Yaskawa INFORM job: DEMO_ROOF_UPPER_0625_3PAINT_6.JBI

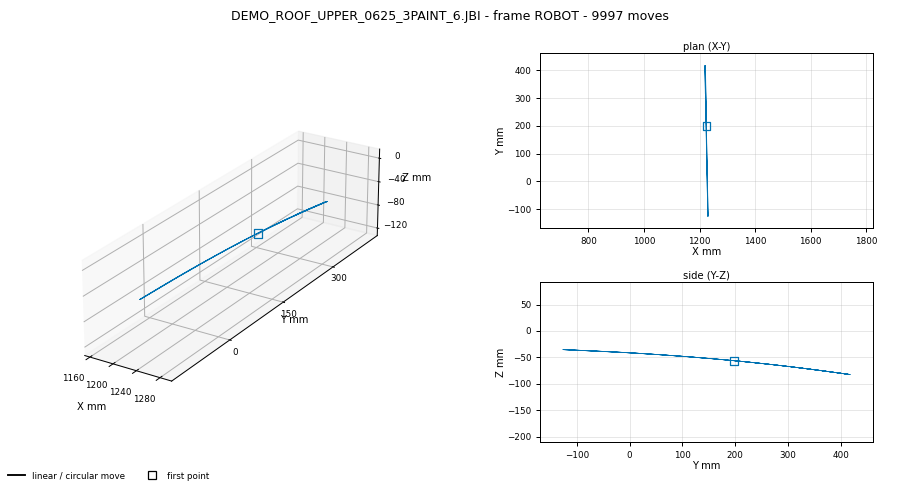
[picture p0: tool path of DEMO_ROOF_UPPER_0625_3PAINT_6.JBI in frame ROBOT, 9997 of 9997 moves have a stored position in this frame; points joined in program order, loops and branches not executed]
/JOB
//NAME DEMO_ROOF_UPPER_0625_3PAINT6
//POS
///NPOS 9997,0,0,0,0,0
///TOOL 0
///USER 0
///POSTYPE ROBOT
///RECTAN
///RCONF 1,0,0,0,0,0,0,0,0,0,0,0,0,0,0,0,0,0,0,0,0,0,0,0
C00000=1225.136,197.844,-56.153,-177.445,6.042,148.322
C00001=1225.132,198.093,-56.176,-177.443,6.043,148.321
C00002=1225.127,198.342,-56.200,-177.440,6.045,148.321
C00003=1225.123,198.590,-56.224,-177.437,6.047,148.321
C00004=1225.118,198.839,-56.247,-177.434,6.049,148.320
C00005=1225.114,199.088,-56.271,-177.432,6.050,148.320
C00006=1225.109,199.337,-56.294,-177.430,6.052,148.319
C00007=1225.104,199.586,-56.318,-177.427,6.053,148.319
C00008=1225.100,199.834,-56.342,-177.424,6.055,148.319
C00009=1225.094,200.083,-56.366,-177.422,6.057,148.318
C00010=1225.090,200.332,-56.390,-177.420,6.058,148.318
C00011=1225.085,200.581,-56.413,-177.417,6.060,148.318
C00012=1225.081,200.829,-56.437,-177.414,6.062,148.317
C00013=1225.077,201.079,-56.461,-177.412,6.064,148.317
C00014=1225.072,201.327,-56.485,-177.409,6.064,148.316
C00015=1225.068,201.577,-56.509,-177.406,6.066,148.316
C00016=1225.063,201.825,-56.533,-177.404,6.068,148.316
C00017=1225.059,202.074,-56.556,-177.401,6.070,148.315
C00018=1225.053,202.323,-56.581,-177.399,6.072,148.315
C00019=1225.049,202.572,-56.604,-177.396,6.073,148.315
C00020=1225.044,202.820,-56.628,-177.394,6.075,148.314
C00021=1225.040,203.069,-56.652,-177.391,6.076,148.314
C00022=1225.036,203.318,-56.676,-177.389,6.078,148.314
C00023=1225.031,203.567,-56.700,-177.386,6.080,148.313
C00024=1225.026,203.816,-56.724,-177.384,6.081,148.313
C00025=1225.022,204.064,-56.748,-177.381,6.083,148.313
C00026=1225.017,204.313,-56.772,-177.378,6.085,148.312
C00027=1225.012,204.562,-56.795,-177.375,6.086,148.312
C00028=1225.008,204.810,-56.819,-177.373,6.088,148.311
C00029=1225.004,205.060,-56.845,-177.370,6.090,148.311
C00030=1224.999,205.309,-56.868,-177.368,6.091,148.311
C00031=1224.994,205.557,-56.892,-177.365,6.093,148.310
C00032=1224.990,205.806,-56.916,-177.363,6.095,148.310
C00033=1224.985,206.055,-56.940,-177.360,6.097,148.310
C00034=1224.980,206.303,-56.964,-177.358,6.099,148.309
C00035=1224.976,206.552,-56.988,-177.355,6.100,148.309
C00036=1224.972,206.801,-57.012,-177.353,6.101,148.309
C00037=1224.967,207.050,-57.037,-177.350,6.103,148.308
C00038=1224.962,207.299,-57.061,-177.348,6.105,148.308
C00039=1224.958,207.547,-57.085,-177.345,6.107,148.308
C00040=1224.953,207.797,-57.109,-177.342,6.109,148.307
C00041=1224.949,208.046,-57.133,-177.340,6.110,148.307
C00042=1224.944,208.294,-57.157,-177.337,6.111,148.306
C00043=1224.940,208.542,-57.181,-177.334,6.113,148.306
C00044=1224.935,208.791,-57.206,-177.332,6.115,148.306
C00045=1224.931,209.040,-57.230,-177.329,6.117,148.305
C00046=1224.926,209.289,-57.254,-177.327,6.119,148.305
C00047=1224.921,209.538,-57.278,-177.324,6.120,148.305
C00048=1224.917,209.786,-57.302,-177.322,6.122,148.304
C00049=1224.912,210.036,-57.327,-177.319,6.124,148.304
C00050=1224.908,210.284,-57.352,-177.317,6.125,148.304
C00051=1224.903,210.533,-57.376,-177.314,6.127,148.303
C00052=1224.898,210.781,-57.400,-177.311,6.129,148.303
C00053=1224.894,211.030,-57.425,-177.309,6.131,148.303
C00054=1224.889,211.301,-57.451,-177.306,6.133,148.302
C00055=1224.884,211.571,-57.477,-177.303,6.135,148.302
C00056=1224.879,211.842,-57.504,-177.300,6.136,148.301
C00057=1224.874,212.111,-57.530,-177.298,6.138,148.301
C00058=1224.870,212.361,-57.555,-177.295,6.140,148.301
C00059=1224.865,212.610,-57.579,-177.292,6.142,148.300
C00060=1224.860,212.859,-57.603,-177.290,6.144,148.300
C00061=1224.856,213.108,-57.628,-177.288,6.145,148.300
C00062=1224.851,213.356,-57.652,-177.285,6.146,148.299
C00063=1224.847,213.604,-57.677,-177.282,6.148,148.299
C00064=1224.842,213.853,-57.702,-177.280,6.150,148.299
C00065=1224.838,214.102,-57.726,-177.277,6.152,148.298
C00066=1224.833,214.351,-57.751,-177.275,6.154,148.298
C00067=1224.828,214.599,-57.775,-177.272,6.156,148.298
C00068=1224.825,214.848,-57.800,-177.269,6.158,148.297
C00069=1224.820,215.097,-57.824,-177.267,6.159,148.297
C00070=1224.814,215.346,-57.849,-177.265,6.161,148.297
C00071=1224.811,215.595,-57.873,-177.262,6.162,148.296
C00072=1224.805,215.844,-57.898,-177.259,6.164,148.296
C00073=1224.801,216.092,-57.922,-177.257,6.166,148.296
C00074=1224.797,216.341,-57.947,-177.254,6.168,148.295
C00075=1224.792,216.589,-57.972,-177.251,6.170,148.295
C00076=1224.788,216.839,-57.997,-177.249,6.172,148.295
C00077=1224.784,217.087,-58.021,-177.246,6.174,148.294
C00078=1224.778,217.336,-58.046,-177.244,6.175,148.294
C00079=1224.774,217.585,-58.071,-177.241,6.176,148.294
C00080=1224.770,217.833,-58.095,-177.239,6.178,148.293
C00081=1224.765,218.082,-58.120,-177.236,6.180,148.293
C00082=1224.761,218.331,-58.145,-177.234,6.182,148.293
C00083=1224.756,218.580,-58.169,-177.231,6.184,148.292
C00084=1224.751,218.828,-58.195,-177.228,6.186,148.292
C00085=1224.747,219.077,-58.219,-177.226,6.188,148.292
C00086=1224.742,219.325,-58.244,-177.223,6.189,148.291
C00087=1224.738,219.575,-58.268,-177.220,6.191,148.291
C00088=1224.733,219.823,-58.294,-177.218,6.192,148.291
C00089=1224.729,220.072,-58.319,-177.216,6.194,148.290
C00090=1224.724,220.321,-58.343,-177.213,6.196,148.290
C00091=1224.720,220.569,-58.368,-177.210,6.198,148.290
C00092=1224.715,220.818,-58.393,-177.208,6.200,148.289
C00093=1224.711,221.066,-58.417,-177.205,6.202,148.289
C00094=1224.706,221.315,-58.443,-177.203,6.203,148.289
C00095=1224.701,221.564,-58.468,-177.200,6.205,148.288
C00096=1224.698,221.813,-58.492,-177.197,6.207,148.288
C00097=1224.693,222.061,-58.517,-177.195,6.209,148.288
C00098=1224.688,222.311,-58.542,-177.192,6.211,148.287
C00099=1224.683,222.559,-58.568,-177.190,6.212,148.287
C00100=1224.680,222.808,-58.592,-177.188,6.214,148.287
C00101=1224.674,223.057,-58.617,-177.185,6.216,148.287
C00102=1224.670,223.305,-58.643,-177.183,6.218,148.286
C00103=1224.665,223.554,-58.667,-177.180,6.220,148.286
C00104=1224.662,223.803,-58.693,-177.177,6.222,148.286
C00105=1224.656,224.051,-58.717,-177.175,6.223,148.285
C00106=1224.652,224.300,-58.743,-177.172,6.225,148.285
C00107=1224.647,224.549,-58.768,-177.169,6.227,148.285
C00108=1224.644,224.797,-58.793,-177.167,6.229,148.284
C00109=1224.638,225.046,-58.817,-177.164,6.231,148.284
C00110=1224.634,225.295,-58.843,-177.162,6.233,148.284
C00111=1224.629,225.544,-58.868,-177.159,6.235,148.283
C00112=1224.625,225.792,-58.894,-177.157,6.236,148.283
C00113=1224.620,226.041,-58.918,-177.154,6.238,148.283
C00114=1224.616,226.290,-58.943,-177.152,6.240,148.283
C00115=1224.611,226.538,-58.969,-177.149,6.242,148.282
C00116=1224.607,226.787,-58.994,-177.147,6.243,148.282
C00117=1224.602,227.035,-59.019,-177.144,6.245,148.282
C00118=1224.598,227.285,-59.044,-177.142,6.247,148.281
C00119=1224.593,227.533,-59.070,-177.139,6.249,148.281
C00120=1224.588,227.782,-59.095,-177.136,6.251,148.281
C00121=1224.585,228.031,-59.120,-177.134,6.253,148.280
C00122=1224.580,228.279,-59.145,-177.131,6.255,148.280
C00123=1224.576,228.528,-59.171,-177.128,6.257,148.280
C00124=1224.571,228.776,-59.196,-177.126,6.258,148.279
C00125=1224.566,229.025,-59.221,-177.124,6.261,148.279
C00126=1224.561,229.273,-59.247,-177.121,6.262,148.279
C00127=1224.557,229.522,-59.273,-177.119,6.263,148.279
C00128=1224.553,229.771,-59.298,-177.116,6.265,148.278
C00129=1224.548,230.020,-59.323,-177.114,6.267,148.278
C00130=1224.544,230.268,-59.349,-177.111,6.269,148.278
C00131=1224.539,230.517,-59.373,-177.109,6.271,148.277
C00132=1224.534,230.766,-59.399,-177.106,6.273,148.277
C00133=1224.530,231.015,-59.425,-177.103,6.275,148.277
C00134=1224.525,231.263,-59.450,-177.101,6.277,148.277
C00135=1224.521,231.512,-59.476,-177.099,6.279,148.276
C00136=1224.516,231.761,-59.501,-177.096,6.281,148.276
C00137=1224.512,232.009,-59.526,-177.093,6.282,148.276
C00138=1224.507,232.258,-59.552,-177.091,6.284,148.275
C00139=1224.503,232.506,-59.578,-177.088,6.286,148.275
C00140=1224.498,232.755,-59.603,-177.085,6.288,148.275
C00141=1224.494,233.004,-59.629,-177.083,6.290,148.274
C00142=1224.489,233.252,-59.654,-177.081,6.292,148.274
C00143=1224.485,233.501,-59.679,-177.078,6.294,148.274
C00144=1224.481,233.750,-59.705,-177.075,6.296,148.274
C00145=1224.476,233.998,-59.731,-177.073,6.298,148.273
C00146=1224.472,234.247,-59.756,-177.070,6.300,148.273
C00147=1224.467,234.496,-59.782,-177.068,6.301,148.273
C00148=1224.462,234.744,-59.808,-177.065,6.304,148.273
C00149=1224.458,234.993,-59.833,-177.063,6.306,148.272
C00150=1224.454,235.241,-59.859,-177.060,6.307,148.272
C00151=1224.450,235.490,-59.885,-177.058,6.309,148.272
C00152=1224.445,235.738,-59.910,-177.055,6.310,148.271
C00153=1224.440,235.987,-59.936,-177.053,6.312,148.271
C00154=1224.436,236.236,-59.962,-177.050,6.314,148.271
C00155=1224.431,236.484,-59.988,-177.048,6.316,148.271
C00156=1224.427,236.733,-60.013,-177.045,6.318,148.270
C00157=1224.423,236.982,-60.039,-177.043,6.320,148.270
C00158=1224.417,237.253,-60.067,-177.040,6.323,148.270
C00159=1224.413,237.524,-60.096,-177.037,6.325,148.269
C00160=1224.408,237.796,-60.123,-177.034,6.326,148.269
C00161=1224.403,238.068,-60.151,-177.032,6.328,148.269
C00162=1224.398,238.316,-60.178,-177.029,6.330,148.268
C00163=1224.394,238.565,-60.204,-177.027,6.332,148.268
C00164=1224.389,238.813,-60.229,-177.024,6.334,148.268
C00165=1224.385,239.062,-60.255,-177.022,6.336,148.268
C00166=1224.381,239.311,-60.281,-177.019,6.338,148.267
C00167=1224.376,239.560,-60.307,-177.017,6.340,148.267
C00168=1224.371,239.808,-60.333,-177.014,6.342,148.267
C00169=1224.367,240.056,-60.359,-177.011,6.344,148.266
C00170=1224.363,240.305,-60.385,-177.009,6.346,148.266
C00171=1224.358,240.554,-60.411,-177.007,6.348,148.266
C00172=1224.354,240.803,-60.437,-177.004,6.350,148.266
C00173=1224.349,241.051,-60.462,-177.001,6.351,148.265
C00174=1224.345,241.299,-60.489,-176.999,6.353,148.265
C00175=1224.340,241.548,-60.515,-176.997,6.355,148.265
C00176=1224.336,241.797,-60.541,-176.994,6.357,148.265
C00177=1224.331,242.046,-60.567,-176.991,6.359,148.264
C00178=1224.326,242.293,-60.593,-176.989,6.361,148.264
C00179=1224.322,242.542,-60.619,-176.986,6.363,148.264
C00180=1224.318,242.791,-60.645,-176.984,6.365,148.264
C00181=1224.313,243.040,-60.672,-176.981,6.367,148.263
C00182=1224.309,243.288,-60.698,-176.978,6.370,148.263
C00183=1224.305,243.537,-60.723,-176.976,6.372,148.263
C00184=1224.299,243.785,-60.750,-176.974,6.374,148.263
C00185=1224.295,244.034,-60.776,-176.971,6.376,148.262
C00186=1224.291,244.283,-60.802,-176.968,6.378,148.262
C00187=1224.286,244.531,-60.829,-176.966,6.379,148.262
C00188=1224.282,244.780,-60.854,-176.963,6.381,148.261
C00189=1224.278,245.029,-60.880,-176.961,6.383,148.261
C00190=1224.273,245.277,-60.907,-176.958,6.385,148.261
C00191=1224.268,245.525,-60.933,-176.956,6.387,148.261
C00192=1224.264,245.774,-60.960,-176.953,6.389,148.260
C00193=1224.259,246.023,-60.985,-176.951,6.391,148.260
C00194=1224.256,246.271,-61.012,-176.948,6.393,148.260
C00195=1224.251,246.520,-61.038,-176.946,6.395,148.260
C00196=1224.247,246.768,-61.065,-176.943,6.397,148.259
C00197=1224.242,247.017,-61.091,-176.941,6.399,148.259
C00198=1224.238,247.265,-61.118,-176.938,6.401,148.259
C00199=1224.233,247.515,-61.144,-176.936,6.403,148.259
C00200=1224.229,247.763,-61.170,-176.933,6.405,148.258
C00201=1224.224,248.011,-61.196,-176.931,6.407,148.258
C00202=1224.219,248.259,-61.223,-176.928,6.409,148.258
C00203=1224.215,248.508,-61.249,-176.926,6.411,148.258
C00204=1224.211,248.757,-61.276,-176.923,6.413,148.257
C00205=1224.206,249.005,-61.301,-176.921,6.415,148.257
C00206=1224.202,249.254,-61.328,-176.918,6.417,148.257
C00207=1224.198,249.502,-61.355,-176.916,6.419,148.257
C00208=1224.193,249.751,-61.381,-176.914,6.421,148.256
C00209=1224.188,250.000,-61.408,-176.910,6.423,148.256
C00210=1224.184,250.249,-61.434,-176.908,6.425,148.256
C00211=1224.179,250.497,-61.461,-176.905,6.427,148.256
C00212=1224.175,250.745,-61.488,-176.903,6.429,148.255
C00213=1224.170,250.994,-61.514,-176.901,6.431,148.255
C00214=1224.166,251.242,-61.540,-176.898,6.433,148.255
C00215=1224.162,251.491,-61.567,-176.896,6.435,148.255
C00216=1224.158,251.740,-61.593,-176.893,6.437,148.254
C00217=1224.153,251.988,-61.620,-176.891,6.439,148.254
C00218=1224.148,252.237,-61.647,-176.888,6.441,148.254
C00219=1224.144,252.485,-61.674,-176.886,6.443,148.254
C00220=1224.139,252.734,-61.700,-176.883,6.445,148.253
C00221=1224.135,252.982,-61.727,-176.881,6.447,148.253
C00222=1224.131,253.231,-61.754,-176.878,6.449,148.253
C00223=1224.126,253.479,-61.781,-176.876,6.451,148.253
C00224=1224.122,253.728,-61.807,-176.873,6.454,148.252
C00225=1224.117,253.977,-61.834,-176.871,6.456,148.252
C00226=1224.113,254.225,-61.861,-176.868,6.458,148.252
C00227=1224.109,254.473,-61.887,-176.865,6.460,148.252
C00228=1224.104,254.722,-61.914,-176.863,6.462,148.251
C00229=1224.099,254.971,-61.941,-176.861,6.464,148.251
C00230=1224.095,255.219,-61.967,-176.858,6.466,148.251
C00231=1224.090,255.468,-61.994,-176.855,6.468,148.251
C00232=1224.086,255.716,-62.021,-176.853,6.470,148.251
C00233=1224.082,255.964,-62.048,-176.851,6.472,148.250
C00234=1224.077,256.213,-62.075,-176.848,6.474,148.250
C00235=1224.073,256.461,-62.102,-176.845,6.477,148.250
C00236=1224.068,256.710,-62.129,-176.843,6.478,148.250
C00237=1224.065,256.959,-62.156,-176.840,6.480,148.249
C00238=1224.060,257.207,-62.183,-176.838,6.482,148.249
C00239=1224.055,257.456,-62.210,-176.835,6.484,148.249
C00240=1224.051,257.704,-62.237,-176.833,6.486,148.249
C00241=1224.046,257.953,-62.263,-176.831,6.488,148.249
C00242=1224.042,258.201,-62.290,-176.828,6.490,148.248
C00243=1224.037,258.450,-62.317,-176.825,6.492,148.248
C00244=1224.032,258.698,-62.344,-176.823,6.494,148.248
C00245=1224.029,258.946,-62.371,-176.820,6.497,148.248
C00246=1224.024,259.194,-62.398,-176.818,6.499,148.248
C00247=1224.020,259.444,-62.425,-176.815,6.501,148.247
C00248=1224.015,259.692,-62.452,-176.813,6.503,148.247
C00249=1224.011,259.941,-62.480,-176.811,6.505,148.247
C00250=1224.006,260.189,-62.507,-176.808,6.507,148.247
C00251=1224.002,260.437,-62.533,-176.805,6.509,148.246
C00252=1223.998,260.686,-62.560,-176.803,6.511,148.246
C00253=1223.993,260.934,-62.587,-176.800,6.514,148.246
C00254=1223.989,261.183,-62.615,-176.798,6.516,148.246
C00255=1223.984,261.432,-62.642,-176.795,6.518,148.246
C00256=1223.980,261.680,-62.669,-176.793,6.520,148.245
C00257=1223.975,261.928,-62.696,-176.791,6.522,148.245
C00258=1223.971,262.177,-62.723,-176.788,6.524,148.245
C00259=1223.967,262.425,-62.750,-176.785,6.526,148.245
C00260=1223.963,262.674,-62.777,-176.783,6.528,148.245
C00261=1223.958,262.923,-62.805,-176.780,6.531,148.244
C00262=1223.953,263.195,-62.835,-176.778,6.533,148.244
C00263=1223.948,263.468,-62.865,-176.775,6.535,148.244
C00264=1223.944,263.740,-62.894,-176.772,6.538,148.244
C00265=1223.938,264.013,-62.925,-176.770,6.540,148.243
C00266=1223.934,264.262,-62.952,-176.767,6.543,148.243
C00267=1223.930,264.510,-62.979,-176.764,6.544,148.243
C00268=1223.925,264.758,-63.007,-176.762,6.546,148.243
C00269=1223.921,265.007,-63.034,-176.760,6.549,148.243
C00270=1223.916,265.255,-63.061,-176.757,6.550,148.242
C00271=1223.912,265.504,-63.088,-176.755,6.553,148.242
C00272=1223.908,265.752,-63.116,-176.752,6.555,148.242
C00273=1223.903,266.001,-63.143,-176.750,6.558,148.242
C00274=1223.899,266.249,-63.171,-176.747,6.559,148.242
C00275=1223.894,266.498,-63.198,-176.744,6.561,148.241
C00276=1223.890,266.746,-63.225,-176.742,6.564,148.241
C00277=1223.885,266.994,-63.253,-176.740,6.565,148.241
C00278=1223.881,267.243,-63.280,-176.738,6.568,148.241
C00279=1223.877,267.492,-63.308,-176.734,6.570,148.241
C00280=1223.872,267.740,-63.336,-176.732,6.573,148.241
C00281=1223.868,267.988,-63.363,-176.730,6.574,148.240
C00282=1223.864,268.237,-63.391,-176.727,6.576,148.240
C00283=1223.859,268.485,-63.418,-176.725,6.579,148.240
C00284=1223.855,268.733,-63.446,-176.722,6.580,148.240
C00285=1223.850,268.982,-63.473,-176.720,6.583,148.240
C00286=1223.846,269.231,-63.501,-176.717,6.585,148.239
C00287=1223.841,269.479,-63.528,-176.715,6.588,148.239
C00288=1223.837,269.727,-63.556,-176.712,6.589,148.239
C00289=1223.833,269.976,-63.584,-176.710,6.592,148.239
C00290=1223.828,270.224,-63.611,-176.708,6.594,148.239
C00291=1223.824,270.472,-63.638,-176.705,6.597,148.239
C00292=1223.820,270.721,-63.667,-176.702,6.598,148.238
C00293=1223.815,270.970,-63.694,-176.700,6.601,148.238
C00294=1223.810,271.218,-63.722,-176.698,6.603,148.238
C00295=1223.807,271.466,-63.750,-176.696,6.605,148.238
C00296=1223.802,271.715,-63.777,-176.692,6.608,148.238
C00297=1223.797,271.963,-63.805,-176.690,6.609,148.237
C00298=1223.793,272.212,-63.832,-176.688,6.612,148.237
C00299=1223.788,272.460,-63.861,-176.685,6.613,148.237
C00300=1223.784,272.708,-63.889,-176.683,6.616,148.237
C00301=1223.780,272.957,-63.916,-176.680,6.618,148.237
C00302=1223.776,273.205,-63.944,-176.678,6.621,148.236
C00303=1223.772,273.454,-63.972,-176.675,6.623,148.236
C00304=1223.766,273.702,-64.000,-176.673,6.625,148.236
C00305=1223.762,273.950,-64.027,-176.671,6.627,148.236
C00306=1223.758,274.199,-64.056,-176.668,6.630,148.236
C00307=1223.754,274.447,-64.083,-176.666,6.632,148.236
C00308=1223.749,274.696,-64.111,-176.663,6.634,148.235
C00309=1223.745,274.944,-64.139,-176.661,6.636,148.235
C00310=1223.741,275.192,-64.167,-176.658,6.638,148.235
C00311=1223.736,275.441,-64.196,-176.656,6.641,148.235
C00312=1223.731,275.689,-64.223,-176.653,6.643,148.235
C00313=1223.728,275.938,-64.251,-176.651,6.645,148.235
C00314=1223.723,276.186,-64.279,-176.648,6.647,148.234
C00315=1223.718,276.434,-64.307,-176.646,6.650,148.234
C00316=1223.714,276.683,-64.335,-176.643,6.652,148.234
C00317=1223.710,276.931,-64.362,-176.641,6.654,148.234
C00318=1223.705,277.180,-64.391,-176.638,6.656,148.234
C00319=1223.701,277.428,-64.419,-176.636,6.658,148.234
C00320=1223.697,277.676,-64.447,-176.633,6.661,148.234
C00321=1223.692,277.925,-64.475,-176.631,6.663,148.233
C00322=1223.688,278.173,-64.503,-176.629,6.665,148.233
C00323=1223.683,278.421,-64.532,-176.626,6.667,148.233
C00324=1223.680,278.670,-64.560,-176.623,6.670,148.233
C00325=1223.675,278.918,-64.588,-176.621,6.672,148.233
C00326=1223.671,279.167,-64.616,-176.619,6.674,148.233
C00327=1223.666,279.415,-64.644,-176.616,6.676,148.232
C00328=1223.662,279.663,-64.673,-176.614,6.679,148.232
C00329=1223.657,279.912,-64.700,-176.611,6.681,148.232
C00330=1223.653,280.161,-64.728,-176.609,6.683,148.232
C00331=1223.648,280.409,-64.756,-176.607,6.686,148.232
C00332=1223.645,280.657,-64.785,-176.604,6.687,148.232
C00333=1223.640,280.905,-64.814,-176.601,6.690,148.231
C00334=1223.636,281.153,-64.842,-176.599,6.693,148.231
C00335=1223.631,281.402,-64.870,-176.597,6.695,148.231
C00336=1223.627,281.650,-64.898,-176.595,6.697,148.231
C00337=1223.622,281.898,-64.927,-176.591,6.700,148.231
C00338=1223.618,282.147,-64.955,-176.589,6.702,148.231
C00339=1223.613,282.395,-64.983,-176.587,6.704,148.231
C00340=1223.610,282.644,-65.011,-176.585,6.706,148.230
C00341=1223.604,282.892,-65.040,-176.582,6.709,148.230
C00342=1223.601,283.141,-65.068,-176.579,6.711,148.230
C00343=1223.596,283.389,-65.097,-176.577,6.713,148.230
C00344=1223.592,283.637,-65.125,-176.575,6.716,148.230
C00345=1223.588,283.886,-65.154,-176.572,6.718,148.230
C00346=1223.583,284.133,-65.182,-176.570,6.720,148.230
C00347=1223.579,284.382,-65.210,-176.568,6.722,148.230
C00348=1223.574,284.630,-65.238,-176.565,6.725,148.229
C00349=1223.570,284.878,-65.268,-176.562,6.727,148.229
C00350=1223.566,285.127,-65.296,-176.560,6.729,148.229
C00351=1223.561,285.375,-65.324,-176.558,6.731,148.229
C00352=1223.557,285.624,-65.353,-176.555,6.734,148.229
C00353=1223.553,285.872,-65.381,-176.553,6.737,148.229
C00354=1223.548,286.120,-65.410,-176.550,6.739,148.229
C00355=1223.544,286.369,-65.439,-176.548,6.741,148.228
C00356=1223.540,286.617,-65.467,-176.546,6.744,148.228
C00357=1223.535,286.865,-65.496,-176.543,6.746,148.228
C00358=1223.531,287.113,-65.524,-176.541,6.748,148.228
C00359=1223.527,287.362,-65.553,-176.538,6.751,148.228
C00360=1223.522,287.610,-65.582,-176.536,6.753,148.228
C00361=1223.518,287.858,-65.610,-176.533,6.755,148.228
C00362=1223.514,288.107,-65.639,-176.531,6.757,148.228
C00363=1223.509,288.355,-65.668,-176.528,6.760,148.227
C00364=1223.505,288.603,-65.696,-176.526,6.762,148.227
C00365=1223.501,288.852,-65.725,-176.524,6.764,148.227
C00366=1223.496,289.126,-65.757,-176.521,6.767,148.227
C00367=1223.491,289.400,-65.789,-176.518,6.770,148.227
C00368=1223.486,289.675,-65.820,-176.516,6.772,148.227
C00369=1223.481,289.948,-65.851,-176.513,6.775,148.227
C00370=1223.477,290.196,-65.881,-176.511,6.777,148.227
C00371=1223.472,290.445,-65.910,-176.508,6.779,148.226
C00372=1223.469,290.693,-65.938,-176.506,6.782,148.226
C00373=1223.464,290.941,-65.967,-176.503,6.784,148.226
C00374=1223.460,291.190,-65.996,-176.501,6.787,148.226
C00375=1223.455,291.439,-66.025,-176.498,6.789,148.226
C00376=1223.451,291.686,-66.054,-176.496,6.792,148.226
C00377=1223.447,291.935,-66.082,-176.494,6.794,148.226
C00378=1223.442,292.183,-66.112,-176.491,6.797,148.226
C00379=1223.438,292.432,-66.140,-176.489,6.799,148.226
C00380=1223.433,292.680,-66.170,-176.487,6.801,148.226
C00381=1223.430,292.927,-66.198,-176.484,6.803,148.225
C00382=1223.425,293.176,-66.227,-176.482,6.806,148.225
C00383=1223.421,293.425,-66.257,-176.479,6.808,148.225
C00384=1223.416,293.673,-66.285,-176.477,6.810,148.225
C00385=1223.412,293.921,-66.314,-176.474,6.813,148.225
C00386=1223.408,294.169,-66.344,-176.472,6.816,148.225
C00387=1223.404,294.418,-66.372,-176.470,6.818,148.225
C00388=1223.399,294.665,-66.401,-176.467,6.821,148.225
C00389=1223.395,294.914,-66.431,-176.465,6.823,148.225
C00390=1223.390,295.163,-66.459,-176.463,6.825,148.225
C00391=1223.386,295.411,-66.489,-176.460,6.828,148.225
C00392=1223.381,295.658,-66.518,-176.458,6.830,148.224
C00393=1223.377,295.907,-66.547,-176.455,6.832,148.224
C00394=1223.373,296.156,-66.576,-176.453,6.835,148.224
C00395=1223.369,296.404,-66.605,-176.451,6.837,148.224
C00396=1223.365,296.652,-66.634,-176.449,6.840,148.224
C00397=1223.360,296.899,-66.663,-176.446,6.843,148.224
C00398=1223.356,297.148,-66.692,-176.443,6.845,148.224
C00399=1223.352,297.397,-66.722,-176.441,6.847,148.224
C00400=1223.348,297.645,-66.751,-176.439,6.850,148.224
C00401=1223.343,297.893,-66.781,-176.436,6.852,148.224
C00402=1223.339,298.141,-66.810,-176.434,6.854,148.224
C00403=1223.334,298.390,-66.838,-176.432,6.857,148.224
C00404=1223.330,298.638,-66.868,-176.429,6.859,148.223
C00405=1223.326,298.886,-66.897,-176.427,6.861,148.223
C00406=1223.322,299.134,-66.927,-176.424,6.865,148.223
C00407=1223.317,299.383,-66.956,-176.422,6.867,148.223
C00408=1223.313,299.631,-66.986,-176.420,6.869,148.223
C00409=1223.308,299.878,-67.015,-176.417,6.872,148.223
C00410=1223.304,300.127,-67.044,-176.415,6.874,148.223
C00411=1223.300,300.375,-67.074,-176.413,6.876,148.223
C00412=1223.296,300.624,-67.102,-176.410,6.879,148.223
C00413=1223.291,300.872,-67.132,-176.408,6.881,148.223
C00414=1223.287,301.120,-67.161,-176.406,6.884,148.223
C00415=1223.283,301.369,-67.191,-176.403,6.887,148.223
C00416=1223.278,301.617,-67.221,-176.401,6.889,148.223
C00417=1223.274,301.866,-67.250,-176.399,6.891,148.223
C00418=1223.269,302.113,-67.279,-176.396,6.894,148.223
C00419=1223.265,302.361,-67.309,-176.394,6.896,148.223
C00420=1223.261,302.610,-67.338,-176.392,6.898,148.222
C00421=1223.257,302.857,-67.368,-176.389,6.901,148.222
C00422=1223.253,303.106,-67.398,-176.387,6.903,148.222
C00423=1223.249,303.354,-67.427,-176.385,6.906,148.222
C00424=1223.244,303.602,-67.457,-176.382,6.909,148.222
C00425=1223.239,303.851,-67.487,-176.380,6.911,148.222
C00426=1223.235,304.099,-67.516,-176.378,6.913,148.222
C00427=1223.231,304.347,-67.546,-176.375,6.916,148.222
C00428=1223.227,304.595,-67.575,-176.373,6.918,148.222
C00429=1223.223,304.844,-67.605,-176.370,6.921,148.222
C00430=1223.218,305.092,-67.634,-176.368,6.924,148.222
C00431=1223.214,305.340,-67.665,-176.366,6.926,148.222
C00432=1223.209,305.588,-67.694,-176.363,6.929,148.222
C00433=1223.205,305.836,-67.723,-176.361,6.931,148.222
C00434=1223.201,306.084,-67.753,-176.359,6.933,148.222
C00435=1223.196,306.333,-67.783,-176.357,6.936,148.222
C00436=1223.192,306.580,-67.813,-176.354,6.939,148.222
C00437=1223.188,306.829,-67.842,-176.352,6.941,148.222
C00438=1223.184,307.077,-67.872,-176.350,6.944,148.222
C00439=1223.179,307.325,-67.902,-176.348,6.946,148.222
C00440=1223.175,307.573,-67.932,-176.345,6.949,148.222
C00441=1223.171,307.821,-67.962,-176.343,6.951,148.222
C00442=1223.166,308.070,-67.991,-176.341,6.954,148.221
C00443=1223.162,308.318,-68.021,-176.338,6.957,148.221
C00444=1223.158,308.566,-68.051,-176.336,6.959,148.221
C00445=1223.153,308.814,-68.081,-176.334,6.961,148.221
C00446=1223.149,309.063,-68.111,-176.331,6.964,148.221
C00447=1223.145,309.310,-68.141,-176.329,6.966,148.221
C00448=1223.140,309.559,-68.170,-176.327,6.969,148.221
C00449=1223.136,309.807,-68.200,-176.324,6.972,148.221
C00450=1223.132,310.055,-68.231,-176.322,6.974,148.221
C00451=1223.128,310.304,-68.260,-176.320,6.977,148.221
C00452=1223.124,310.551,-68.291,-176.317,6.979,148.221
C00453=1223.119,310.800,-68.321,-176.315,6.981,148.221
C00454=1223.115,311.048,-68.350,-176.313,6.984,148.221
C00455=1223.111,311.296,-68.381,-176.311,6.987,148.221
C00456=1223.106,311.544,-68.410,-176.308,6.989,148.221
C00457=1223.102,311.792,-68.440,-176.306,6.992,148.221
C00458=1223.098,312.041,-68.471,-176.304,6.994,148.221
C00459=1223.094,312.288,-68.501,-176.301,6.997,148.221
C00460=1223.089,312.537,-68.531,-176.299,7.000,148.221
C00461=1223.085,312.785,-68.561,-176.297,7.002,148.221
C00462=1223.081,313.033,-68.590,-176.295,7.005,148.221
C00463=1223.077,313.282,-68.622,-176.292,7.007,148.221
C00464=1223.072,313.530,-68.651,-176.290,7.009,148.221
C00465=1223.068,313.778,-68.682,-176.288,7.012,148.221
C00466=1223.064,314.025,-68.712,-176.286,7.015,148.221
C00467=1223.059,314.274,-68.742,-176.283,7.018,148.221
C00468=1223.055,314.522,-68.772,-176.281,7.020,148.221
C00469=1223.050,314.770,-68.802,-176.279,7.022,148.221
C00470=1223.046,315.046,-68.836,-176.277,7.026,148.221
C00471=1223.041,315.322,-68.869,-176.274,7.029,148.221
C00472=1223.037,315.598,-68.903,-176.271,7.032,148.221
C00473=1223.031,315.873,-68.936,-176.269,7.034,148.221
C00474=1223.027,316.122,-68.967,-176.266,7.037,148.221
C00475=1223.024,316.370,-68.998,-176.264,7.039,148.221
C00476=1223.019,316.618,-69.028,-176.262,7.042,148.221
C00477=1223.015,316.866,-69.058,-176.260,7.045,148.221
C00478=1223.010,317.114,-69.089,-176.258,7.047,148.221
C00479=1223.006,317.362,-69.118,-176.255,7.050,148.221
C00480=1223.002,317.611,-69.149,-176.253,7.052,148.221
C00481=1222.998,317.858,-69.179,-176.251,7.055,148.221
C00482=1222.993,318.106,-69.210,-176.249,7.058,148.221
C00483=1222.989,318.355,-69.240,-176.247,7.060,148.221
C00484=1222.985,318.602,-69.270,-176.244,7.063,148.221
C00485=1222.981,318.851,-69.301,-176.242,7.065,148.221
C00486=1222.977,319.099,-69.332,-176.240,7.068,148.221
C00487=1222.972,319.347,-69.362,-176.238,7.071,148.221
C00488=1222.968,319.594,-69.393,-176.236,7.073,148.221
C00489=1222.963,319.843,-69.423,-176.233,7.076,148.221
C00490=1222.959,320.092,-69.454,-176.231,7.079,148.221
C00491=1222.955,320.339,-69.484,-176.229,7.081,148.221
C00492=1222.951,320.587,-69.515,-176.227,7.084,148.221
C00493=1222.946,320.835,-69.545,-176.224,7.086,148.221
C00494=1222.943,321.084,-69.576,-176.222,7.089,148.221
C00495=1222.938,321.332,-69.607,-176.220,7.092,148.221
C00496=1222.934,321.579,-69.637,-176.218,7.094,148.221
C00497=1222.930,321.828,-69.667,-176.215,7.097,148.221
C00498=1222.926,322.076,-69.698,-176.214,7.099,148.222
C00499=1222.921,322.324,-69.729,-176.211,7.103,148.222
C00500=1222.917,322.572,-69.759,-176.209,7.105,148.222
C00501=1222.913,322.821,-69.790,-176.207,7.107,148.222
C00502=1222.908,323.069,-69.821,-176.205,7.110,148.222
C00503=1222.904,323.317,-69.852,-176.203,7.113,148.222
C00504=1222.900,323.564,-69.882,-176.200,7.116,148.222
C00505=1222.896,323.813,-69.913,-176.198,7.118,148.222
C00506=1222.891,324.061,-69.944,-176.196,7.120,148.222
C00507=1222.887,324.308,-69.974,-176.194,7.124,148.222
C00508=1222.883,324.557,-70.005,-176.192,7.126,148.222
C00509=1222.879,324.805,-70.036,-176.190,7.128,148.222
C00510=1222.875,325.052,-70.067,-176.188,7.132,148.222
C00511=1222.871,325.301,-70.098,-176.186,7.134,148.222
C00512=1222.867,325.549,-70.129,-176.183,7.137,148.222
C00513=1222.862,325.797,-70.159,-176.181,7.139,148.222
C00514=1222.858,326.045,-70.190,-176.179,7.142,148.222
C00515=1222.853,326.293,-70.221,-176.177,7.145,148.222
C00516=1222.849,326.541,-70.252,-176.175,7.147,148.222
C00517=1222.846,326.790,-70.282,-176.172,7.150,148.222
C00518=1222.841,327.037,-70.314,-176.171,7.153,148.223
C00519=1222.837,327.285,-70.345,-176.168,7.155,148.223
C00520=1222.833,327.534,-70.376,-176.166,7.158,148.223
C00521=1222.828,327.782,-70.407,-176.164,7.161,148.223
C00522=1222.823,328.030,-70.437,-176.162,7.164,148.223
C00523=1222.820,328.277,-70.469,-176.160,7.166,148.223
C00524=1222.816,328.525,-70.499,-176.158,7.168,148.223
C00525=1222.811,328.773,-70.530,-176.156,7.172,148.223
C00526=1222.807,329.022,-70.561,-176.153,7.174,148.223
C00527=1222.803,329.269,-70.593,-176.151,7.177,148.223
C00528=1222.799,329.518,-70.624,-176.149,7.179,148.223
C00529=1222.794,329.766,-70.655,-176.148,7.182,148.223
C00530=1222.790,330.014,-70.685,-176.145,7.185,148.223
C00531=1222.786,330.262,-70.717,-176.143,7.188,148.224
C00532=1222.781,330.510,-70.748,-176.141,7.190,148.224
C00533=1222.777,330.758,-70.779,-176.139,7.193,148.224
C00534=1222.773,331.006,-70.811,-176.137,7.195,148.224
C00535=1222.768,331.254,-70.841,-176.135,7.199,148.224
C00536=1222.765,331.502,-70.873,-176.133,7.201,148.224
C00537=1222.760,331.750,-70.904,-176.131,7.203,148.224
C00538=1222.757,331.998,-70.935,-176.128,7.207,148.224
C00539=1222.752,332.245,-70.966,-176.127,7.209,148.224
C00540=1222.748,332.494,-70.997,-176.124,7.212,148.224
C00541=1222.744,332.741,-71.029,-176.122,7.215,148.224
C00542=1222.740,332.989,-71.059,-176.120,7.217,148.224
C00543=1222.735,333.238,-71.091,-176.118,7.220,148.225
C00544=1222.730,333.486,-71.123,-176.116,7.223,148.225
C00545=1222.726,333.734,-71.154,-176.114,7.225,148.225
C00546=1222.722,333.982,-71.185,-176.112,7.228,148.225
C00547=1222.718,334.230,-71.216,-176.110,7.231,148.225
C00548=1222.714,334.478,-71.248,-176.108,7.234,148.225
C00549=1222.710,334.726,-71.279,-176.106,7.236,148.225
C00550=1222.705,334.974,-71.310,-176.104,7.239,148.225
C00551=1222.701,335.222,-71.342,-176.102,7.242,148.226
C00552=1222.697,335.470,-71.373,-176.100,7.244,148.225
C00553=1222.693,335.718,-71.404,-176.098,7.248,148.226
C00554=1222.689,335.966,-71.436,-176.096,7.250,148.226
C00555=1222.685,336.214,-71.468,-176.094,7.252,148.226
C00556=1222.681,336.462,-71.498,-176.092,7.256,148.226
C00557=1222.677,336.710,-71.530,-176.090,7.258,148.226
C00558=1222.671,336.958,-71.561,-176.088,7.260,148.226
C00559=1222.668,337.206,-71.593,-176.086,7.264,148.226
C00560=1222.663,337.453,-71.625,-176.084,7.266,148.227
C00561=1222.659,337.702,-71.656,-176.082,7.269,148.227
C00562=1222.655,337.949,-71.687,-176.080,7.272,148.227
C00563=1222.651,338.197,-71.719,-176.078,7.274,148.227
C00564=1222.647,338.445,-71.750,-176.076,7.278,148.227
C00565=1222.642,338.694,-71.782,-176.074,7.280,148.227
C00566=1222.639,338.942,-71.814,-176.072,7.283,148.227
C00567=1222.634,339.190,-71.845,-176.070,7.286,148.227
C00568=1222.630,339.438,-71.877,-176.068,7.288,148.228
C00569=1222.626,339.685,-71.908,-176.066,7.291,148.228
C00570=1222.622,339.933,-71.941,-176.064,7.294,148.228
C00571=1222.617,340.181,-71.972,-176.062,7.296,148.228
C00572=1222.613,340.429,-72.003,-176.060,7.300,148.228
C00573=1222.609,340.677,-72.035,-176.058,7.302,148.228
C00574=1222.604,340.955,-72.071,-176.056,7.305,148.229
C00575=1222.599,341.233,-72.106,-176.054,7.308,148.229
C00576=1222.595,341.510,-72.142,-176.052,7.311,148.229
C00577=1222.590,341.788,-72.178,-176.050,7.314,148.229
C00578=1222.586,342.037,-72.209,-176.048,7.317,148.229
C00579=1222.582,342.284,-72.240,-176.045,7.320,148.229
C00580=1222.578,342.532,-72.272,-176.044,7.323,148.229
C00581=1222.573,342.780,-72.305,-176.042,7.325,148.230
C00582=1222.569,343.028,-72.336,-176.040,7.328,148.230
C00583=1222.565,343.276,-72.368,-176.038,7.331,148.230
C00584=1222.560,343.523,-72.400,-176.037,7.333,148.230
C00585=1222.557,343.771,-72.432,-176.034,7.337,148.230
C00586=1222.553,344.020,-72.464,-176.032,7.339,148.230
C00587=1222.548,344.268,-72.495,-176.030,7.342,148.231
C00588=1222.544,344.516,-72.527,-176.029,7.345,148.231
C00589=1222.540,344.764,-72.559,-176.027,7.347,148.231
C00590=1222.535,345.012,-72.591,-176.025,7.351,148.231
C00591=1222.531,345.260,-72.623,-176.023,7.353,148.231
C00592=1222.527,345.507,-72.654,-176.021,7.356,148.232
C00593=1222.523,345.755,-72.687,-176.019,7.359,148.232
C00594=1222.519,346.003,-72.719,-176.017,7.361,148.232
C00595=1222.514,346.251,-72.751,-176.016,7.364,148.232
C00596=1222.510,346.499,-72.782,-176.013,7.367,148.232
C00597=1222.507,346.747,-72.814,-176.012,7.370,148.232
C00598=1222.501,346.995,-72.846,-176.010,7.372,148.232
C00599=1222.498,347.242,-72.879,-176.008,7.376,148.233
C00600=1222.494,347.490,-72.911,-176.006,7.378,148.233
C00601=1222.490,347.738,-72.943,-176.005,7.381,148.233
C00602=1222.485,347.986,-72.975,-176.002,7.384,148.233
C00603=1222.481,348.234,-73.007,-176.001,7.387,148.233
C00604=1222.477,348.482,-73.039,-175.999,7.389,148.234
C00605=1222.472,348.730,-73.071,-175.997,7.393,148.234
C00606=1222.469,348.978,-73.103,-175.995,7.395,148.234
C00607=1222.464,349.226,-73.135,-175.994,7.398,148.234
C00608=1222.460,349.473,-73.168,-175.992,7.401,148.234
C00609=1222.456,349.721,-73.200,-175.990,7.404,148.235
C00610=1222.452,349.969,-73.232,-175.988,7.406,148.235
C00611=1222.448,350.218,-73.264,-175.987,7.409,148.235
C00612=1222.443,350.465,-73.296,-175.984,7.412,148.235
C00613=1222.439,350.713,-73.329,-175.983,7.414,148.235
C00614=1222.436,350.961,-73.361,-175.981,7.417,148.236
C00615=1222.431,351.209,-73.393,-175.979,7.420,148.236
C00616=1222.427,351.456,-73.425,-175.977,7.423,148.236
C00617=1222.423,351.704,-73.458,-175.976,7.425,148.236
C00618=1222.419,351.952,-73.490,-175.974,7.429,148.236
C00619=1222.415,352.201,-73.522,-175.972,7.431,148.237
C00620=1222.409,352.448,-73.554,-175.971,7.434,148.237
C00621=1222.406,352.696,-73.587,-175.969,7.437,148.237
C00622=1222.402,352.944,-73.619,-175.967,7.440,148.237
C00623=1222.398,353.192,-73.651,-175.965,7.443,148.238
C00624=1222.394,353.440,-73.684,-175.964,7.445,148.238
C00625=1222.389,353.687,-73.716,-175.961,7.448,148.238
C00626=1222.385,353.935,-73.748,-175.960,7.451,148.238
C00627=1222.381,354.183,-73.781,-175.959,7.454,148.239
C00628=1222.377,354.431,-73.813,-175.956,7.457,148.239
C00629=1222.373,354.680,-73.846,-175.955,7.460,148.239
C00630=1222.369,354.926,-73.878,-175.953,7.462,148.239
C00631=1222.364,355.175,-73.910,-175.952,7.465,148.239
C00632=1222.360,355.422,-73.943,-175.949,7.468,148.240
C00633=1222.356,355.670,-73.975,-175.948,7.471,148.240
C00634=1222.352,355.919,-74.008,-175.947,7.473,148.240
C00635=1222.347,356.166,-74.040,-175.945,7.476,148.240
C00636=1222.344,356.414,-74.072,-175.943,7.479,148.241
C00637=1222.339,356.662,-74.105,-175.942,7.482,148.241
C00638=1222.335,356.910,-74.138,-175.940,7.485,148.241
C00639=1222.332,357.157,-74.170,-175.938,7.488,148.241
C00640=1222.327,357.406,-74.203,-175.936,7.491,148.242
C00641=1222.323,357.653,-74.236,-175.935,7.493,148.242
C00642=1222.319,357.901,-74.268,-175.933,7.496,148.242
C00643=1222.315,358.148,-74.301,-175.931,7.499,148.242
C00644=1222.310,358.397,-74.333,-175.930,7.502,148.243
C00645=1222.306,358.645,-74.366,-175.928,7.505,148.243
C00646=1222.302,358.893,-74.398,-175.927,7.507,148.243
C00647=1222.298,359.140,-74.431,-175.924,7.510,148.243
C00648=1222.294,359.388,-74.464,-175.923,7.513,148.244
C00649=1222.290,359.635,-74.496,-175.922,7.516,148.244
C00650=1222.286,359.883,-74.529,-175.920,7.518,148.244
C00651=1222.281,360.131,-74.561,-175.919,7.521,148.245
C00652=1222.277,360.379,-74.595,-175.917,7.524,148.245
C00653=1222.273,360.627,-74.628,-175.915,7.527,148.245
C00654=1222.269,360.875,-74.660,-175.914,7.530,148.245
C00655=1222.265,361.123,-74.693,-175.912,7.532,148.246
C00656=1222.261,361.370,-74.726,-175.910,7.536,148.246
C00657=1222.256,361.619,-74.758,-175.909,7.539,148.246
C00658=1222.253,361.866,-74.791,-175.908,7.541,148.247
C00659=1222.249,362.114,-74.824,-175.906,7.544,148.247
C00660=1222.244,362.362,-74.856,-175.904,7.546,148.247
C00661=1222.240,362.609,-74.889,-175.903,7.550,148.247
C00662=1222.236,362.857,-74.923,-175.901,7.553,148.248
C00663=1222.231,363.105,-74.956,-175.900,7.555,148.248
C00664=1222.228,363.353,-74.988,-175.898,7.558,148.248
C00665=1222.224,363.601,-75.021,-175.897,7.561,148.249
C00666=1222.219,363.848,-75.054,-175.895,7.564,148.249
C00667=1222.215,364.096,-75.087,-175.894,7.567,148.249
C00668=1222.211,364.344,-75.119,-175.892,7.569,148.249
C00669=1222.207,364.592,-75.153,-175.891,7.572,148.250
C00670=1222.203,364.839,-75.185,-175.889,7.575,148.250
C00671=1222.199,365.087,-75.218,-175.888,7.578,148.250
C00672=1222.195,365.335,-75.251,-175.886,7.581,148.251
C00673=1222.191,365.583,-75.284,-175.885,7.584,148.251
C00674=1222.186,365.831,-75.317,-175.883,7.586,148.251
C00675=1222.182,366.079,-75.350,-175.882,7.589,148.252
C00676=1222.178,366.326,-75.383,-175.881,7.592,148.252
C00677=1222.174,366.574,-75.417,-175.879,7.595,148.252
C00678=1222.169,366.854,-75.453,-175.877,7.598,148.253
C00679=1222.165,367.134,-75.491,-175.876,7.601,148.253
C00680=1222.160,367.414,-75.528,-175.874,7.604,148.253
C00681=1222.155,367.694,-75.565,-175.873,7.607,148.254
C00682=1222.151,367.942,-75.598,-175.871,7.611,148.254
C00683=1222.147,368.189,-75.632,-175.869,7.613,148.254
C00684=1222.143,368.437,-75.664,-175.868,7.616,148.255
C00685=1222.139,368.684,-75.697,-175.867,7.619,148.255
C00686=1222.135,368.932,-75.730,-175.865,7.622,148.255
C00687=1222.131,369.180,-75.764,-175.864,7.624,148.256
C00688=1222.127,369.428,-75.797,-175.863,7.627,148.256
C00689=1222.123,369.675,-75.830,-175.862,7.630,148.256
C00690=1222.119,369.923,-75.863,-175.860,7.633,148.257
C00691=1222.114,370.171,-75.896,-175.859,7.635,148.257
C00692=1222.110,370.419,-75.929,-175.858,7.638,148.257
C00693=1222.106,370.666,-75.962,-175.856,7.641,148.258
C00694=1222.102,370.914,-75.996,-175.855,7.644,148.258
C00695=1222.098,371.162,-76.029,-175.853,7.647,148.258
C00696=1222.093,371.410,-76.063,-175.852,7.650,148.259
C00697=1222.089,371.657,-76.096,-175.851,7.653,148.259
C00698=1222.085,371.906,-76.129,-175.849,7.655,148.259
C00699=1222.081,372.154,-76.162,-175.848,7.658,148.260
C00700=1222.077,372.401,-76.196,-175.847,7.661,148.260
C00701=1222.073,372.648,-76.229,-175.845,7.663,148.260
C00702=1222.069,372.896,-76.263,-175.844,7.666,148.261
C00703=1222.065,373.144,-76.296,-175.843,7.669,148.261
C00704=1222.061,373.392,-76.329,-175.842,7.672,148.262
C00705=1222.057,373.639,-76.362,-175.841,7.675,148.262
C00706=1222.052,373.887,-76.395,-175.840,7.678,148.262
C00707=1222.048,374.135,-76.428,-175.838,7.680,148.263
C00708=1222.044,374.383,-76.461,-175.837,7.683,148.263
C00709=1222.040,374.630,-76.495,-175.836,7.686,148.263
C00710=1222.036,374.878,-76.529,-175.834,7.689,148.264
C00711=1222.032,375.126,-76.563,-175.833,7.691,148.264
C00712=1222.028,375.374,-76.596,-175.833,7.693,148.265
C00713=1222.024,375.622,-76.629,-175.831,7.696,148.265
C00714=1222.020,375.869,-76.663,-175.830,7.699,148.265
C00715=1222.016,376.116,-76.696,-175.829,7.702,148.266
C00716=1222.012,376.364,-76.729,-175.827,7.704,148.266
C00717=1222.007,376.612,-76.763,-175.826,7.707,148.266
C00718=1222.003,376.860,-76.796,-175.825,7.710,148.267
C00719=1221.999,377.108,-76.830,-175.824,7.713,148.267
C00720=1221.995,377.355,-76.863,-175.823,7.716,148.267
C00721=1221.991,377.603,-76.897,-175.822,7.718,148.268
C00722=1221.987,377.851,-76.930,-175.820,7.721,148.268
C00723=1221.982,378.098,-76.964,-175.819,7.724,148.269
C00724=1221.978,378.346,-76.997,-175.819,7.726,148.269
C00725=1221.974,378.594,-77.031,-175.817,7.729,148.269
C00726=1221.971,378.842,-77.065,-175.816,7.732,148.270
C00727=1221.967,379.089,-77.098,-175.815,7.735,148.270
C00728=1221.962,379.337,-77.132,-175.814,7.737,148.271
C00729=1221.958,379.585,-77.166,-175.813,7.740,148.271
C00730=1221.954,379.832,-77.199,-175.811,7.743,148.271
C00731=1221.950,380.080,-77.232,-175.810,7.746,148.272
C00732=1221.946,380.328,-77.267,-175.810,7.748,148.272
C00733=1221.942,380.576,-77.300,-175.808,7.751,148.273
C00734=1221.937,380.824,-77.333,-175.807,7.753,148.273
C00735=1221.934,381.071,-77.367,-175.806,7.756,148.273
C00736=1221.929,381.319,-77.401,-175.805,7.759,148.274
C00737=1221.925,381.566,-77.434,-175.804,7.762,148.274
C00738=1221.921,381.814,-77.468,-175.804,7.764,148.275
C00739=1221.917,382.062,-77.501,-175.802,7.767,148.275
C00740=1221.913,382.309,-77.536,-175.801,7.770,148.275
C00741=1221.909,382.557,-77.569,-175.800,7.773,148.276
C00742=1221.905,382.804,-77.603,-175.799,7.775,148.276
C00743=1221.901,383.053,-77.636,-175.798,7.777,148.277
C00744=1221.897,383.300,-77.671,-175.797,7.780,148.277
C00745=1221.892,383.548,-77.704,-175.796,7.783,148.277
C00746=1221.888,383.796,-77.737,-175.795,7.786,148.278
C00747=1221.884,384.043,-77.771,-175.794,7.788,148.278
C00748=1221.880,384.291,-77.805,-175.793,7.791,148.279
C00749=1221.876,384.538,-77.839,-175.792,7.794,148.279
C00750=1221.871,384.787,-77.873,-175.791,7.797,148.280
C00751=1221.868,385.034,-77.906,-175.790,7.799,148.280
C00752=1221.864,385.281,-77.940,-175.790,7.802,148.280
C00753=1221.860,385.529,-77.974,-175.788,7.805,148.281
C00754=1221.856,385.777,-78.008,-175.788,7.807,148.281
C00755=1221.852,386.024,-78.041,-175.787,7.809,148.282
C00756=1221.847,386.272,-78.076,-175.785,7.812,148.282
C00757=1221.843,386.520,-78.109,-175.784,7.815,148.282
C00758=1221.840,386.767,-78.143,-175.784,7.817,148.283
C00759=1221.835,387.015,-78.177,-175.783,7.820,148.283
C00760=1221.831,387.262,-78.211,-175.782,7.823,148.284
C00761=1221.827,387.511,-78.245,-175.781,7.825,148.284
C00762=1221.823,387.758,-78.279,-175.780,7.828,148.285
C00763=1221.819,388.005,-78.313,-175.779,7.831,148.285
C00764=1221.814,388.253,-78.347,-175.778,7.833,148.285
C00765=1221.811,388.501,-78.381,-175.777,7.836,148.286
C00766=1221.806,388.749,-78.415,-175.776,7.838,148.286
C00767=1221.802,388.996,-78.448,-175.776,7.841,148.287
C00768=1221.798,389.243,-78.482,-175.775,7.843,148.287
C00769=1221.794,389.492,-78.516,-175.774,7.845,148.287
C00770=1221.790,389.739,-78.550,-175.773,7.849,148.288
C00771=1221.786,389.987,-78.585,-175.772,7.851,148.288
C00772=1221.782,390.235,-78.618,-175.772,7.853,148.289
C00773=1221.778,390.482,-78.652,-175.770,7.856,148.289
C00774=1221.774,390.730,-78.687,-175.770,7.858,148.290
C00775=1221.770,390.977,-78.720,-175.769,7.861,148.290
C00776=1221.766,391.226,-78.755,-175.768,7.864,148.291
C00777=1221.762,391.473,-78.788,-175.767,7.866,148.291
C00778=1221.757,391.720,-78.823,-175.766,7.869,148.291
C00779=1221.754,391.969,-78.856,-175.766,7.871,148.292
C00780=1221.749,392.216,-78.891,-175.765,7.874,148.292
C00781=1221.745,392.463,-78.925,-175.764,7.876,148.293
C00782=1221.741,392.745,-78.963,-175.763,7.879,148.293
C00783=1221.736,393.027,-79.002,-175.763,7.882,148.294
C00784=1221.732,393.309,-79.041,-175.761,7.885,148.294
C00785=1221.727,393.590,-79.080,-175.761,7.888,148.295
C00786=1221.723,393.837,-79.114,-175.760,7.890,148.295
C00787=1221.719,394.085,-79.149,-175.759,7.893,148.296
C00788=1221.715,394.333,-79.182,-175.758,7.896,148.296
C00789=1221.710,394.581,-79.216,-175.757,7.898,148.296
C00790=1221.707,394.828,-79.251,-175.756,7.901,148.297
C00791=1221.702,395.076,-79.285,-175.756,7.903,148.297
C00792=1221.699,395.323,-79.319,-175.755,7.905,148.298
C00793=1221.694,395.572,-79.353,-175.754,7.908,148.298
C00794=1221.690,395.819,-79.387,-175.754,7.910,148.299
C00795=1221.686,396.066,-79.421,-175.753,7.913,148.299
C00796=1221.682,396.314,-79.456,-175.752,7.915,148.299
C00797=1221.678,396.561,-79.490,-175.752,7.918,148.300
C00798=1221.674,396.810,-79.525,-175.751,7.920,148.300
C00799=1221.670,397.057,-79.558,-175.750,7.923,148.301
C00800=1221.665,397.305,-79.592,-175.750,7.925,148.301
C00801=1221.662,397.553,-79.627,-175.748,7.928,148.302
C00802=1221.658,397.800,-79.661,-175.748,7.930,148.302
C00803=1221.654,398.047,-79.695,-175.748,7.932,148.303
C00804=1221.650,398.295,-79.730,-175.746,7.935,148.303
C00805=1221.645,398.543,-79.764,-175.746,7.937,148.304
C00806=1221.641,398.790,-79.798,-175.745,7.940,148.304
C00807=1221.637,399.038,-79.833,-175.745,7.942,148.304
C00808=1221.633,399.286,-79.866,-175.744,7.944,148.305
C00809=1221.629,399.534,-79.901,-175.743,7.947,148.305
C00810=1221.625,399.781,-79.936,-175.743,7.949,148.306
C00811=1221.621,400.028,-79.969,-175.742,7.952,148.306
C00812=1221.617,400.276,-80.004,-175.741,7.955,148.307
C00813=1221.613,400.523,-80.038,-175.741,7.957,148.307
C00814=1221.609,400.771,-80.073,-175.740,7.959,148.307
C00815=1221.605,401.019,-80.107,-175.739,7.962,148.308
C00816=1221.601,401.266,-80.141,-175.739,7.964,148.308
C00817=1221.597,401.514,-80.176,-175.738,7.967,148.309
C00818=1221.593,401.761,-80.210,-175.737,7.969,148.309
C00819=1221.588,402.009,-80.244,-175.737,7.971,148.310
C00820=1221.584,402.257,-80.279,-175.736,7.974,148.310
C00821=1221.581,402.504,-80.313,-175.735,7.976,148.311
C00822=1221.577,402.752,-80.348,-175.735,7.978,148.311
C00823=1221.572,403.000,-80.382,-175.734,7.981,148.311
C00824=1221.568,403.247,-80.416,-175.733,7.983,148.312
C00825=1221.564,403.495,-80.451,-175.733,7.985,148.312
C00826=1221.560,403.742,-80.486,-175.733,7.987,148.313
C00827=1221.556,403.990,-80.520,-175.732,7.990,148.313
C00828=1221.552,404.237,-80.554,-175.731,7.992,148.314
C00829=1221.548,404.486,-80.589,-175.731,7.994,148.314
C00830=1221.544,404.733,-80.623,-175.730,7.997,148.315
C00831=1221.539,404.980,-80.657,-175.729,7.999,148.315
C00832=1221.536,405.228,-80.693,-175.729,8.001,148.315
C00833=1221.532,405.475,-80.727,-175.728,8.003,148.316
C00834=1221.528,405.723,-80.762,-175.728,8.007,148.316
C00835=1221.523,405.970,-80.796,-175.727,8.009,148.317
C00836=1221.520,406.218,-80.830,-175.727,8.011,148.317
C00837=1221.516,406.465,-80.865,-175.726,8.013,148.318
C00838=1221.511,406.713,-80.899,-175.725,8.016,148.318
C00839=1221.507,406.961,-80.934,-175.725,8.018,148.319
C00840=1221.503,407.208,-80.968,-175.724,8.020,148.319
C00841=1221.499,407.456,-81.003,-175.724,8.022,148.319
C00842=1221.495,407.703,-81.038,-175.723,8.024,148.320
C00843=1221.492,407.951,-81.072,-175.722,8.027,148.320
C00844=1221.487,408.198,-81.107,-175.722,8.029,148.321
C00845=1221.483,408.446,-81.142,-175.721,8.031,148.321
C00846=1221.479,408.694,-81.176,-175.721,8.033,148.322
C00847=1221.475,408.942,-81.210,-175.720,8.035,148.322
C00848=1221.471,409.188,-81.245,-175.720,8.039,148.323
C00849=1221.467,409.436,-81.280,-175.719,8.041,148.323
C00850=1221.463,409.684,-81.315,-175.718,8.042,148.323
C00851=1221.459,409.931,-81.349,-175.718,8.045,148.324
C00852=1221.455,410.179,-81.383,-175.718,8.047,148.324
C00853=1221.450,410.427,-81.418,-175.717,8.049,148.325
C00854=1221.447,410.674,-81.454,-175.716,8.052,148.325
C00855=1221.443,410.921,-81.487,-175.716,8.054,148.326
C00856=1221.439,411.169,-81.522,-175.715,8.056,148.326
C00857=1221.434,411.417,-81.557,-175.715,8.058,148.326
C00858=1221.431,411.664,-81.592,-175.714,8.060,148.327
C00859=1221.426,411.912,-81.627,-175.714,8.062,148.327
C00860=1221.423,412.159,-81.661,-175.714,8.065,148.328
C00861=1221.418,412.407,-81.695,-175.712,8.067,148.328
C00862=1221.415,412.654,-81.731,-175.712,8.069,148.328
C00863=1221.410,412.902,-81.765,-175.712,8.072,148.329
C00864=1221.406,413.150,-81.800,-175.711,8.074,148.329
C00865=1221.402,413.397,-81.834,-175.711,8.076,148.330
C00866=1221.399,413.644,-81.870,-175.710,8.078,148.330
C00867=1221.394,413.892,-81.904,-175.709,8.080,148.330
C00868=1221.390,414.140,-81.939,-175.709,8.082,148.331
C00869=1221.385,414.387,-81.973,-175.709,8.084,148.331
C00870=1221.382,414.635,-82.008,-175.708,8.086,148.332
C00871=1221.378,414.882,-82.043,-175.707,8.089,148.332
C00872=1221.374,415.130,-82.078,-175.707,8.091,148.333
C00873=1221.370,415.377,-82.113,-175.706,8.093,148.333
C00874=1221.367,415.592,-82.143,-175.706,8.095,148.333
C00875=1221.363,415.806,-82.173,-175.706,8.097,148.334
C00876=1221.359,416.019,-82.203,-175.706,8.099,148.334
C00877=1221.356,416.234,-82.233,-175.705,8.101,148.335
C00878=1221.353,416.448,-82.263,-175.704,8.103,148.335
C00879=1221.349,416.663,-82.294,-175.704,8.104,148.335
C00880=1221.346,416.876,-82.323,-175.703,8.106,148.336
C00881=1221.346,417.091,-82.353,-175.703,8.108,148.336
C00882=1220.924,417.090,-82.387,-175.706,8.118,148.340
C00883=1220.924,416.875,-82.358,-175.707,8.116,148.339
C00884=1220.927,416.660,-82.327,-175.708,8.114,148.339
C00885=1220.931,416.444,-82.297,-175.708,8.113,148.339
C00886=1220.934,416.229,-82.267,-175.708,8.111,148.338
C00887=1220.937,416.013,-82.236,-175.708,8.109,148.338
C00888=1220.941,415.798,-82.206,-175.709,8.107,148.338
C00889=1220.944,415.582,-82.176,-175.710,8.105,148.337
C00890=1220.948,415.367,-82.146,-175.709,8.104,148.337
C00891=1220.952,415.119,-82.111,-175.710,8.102,148.336
C00892=1220.956,414.872,-82.075,-175.711,8.099,148.336
C00893=1220.961,414.624,-82.041,-175.711,8.097,148.335
C00894=1220.964,414.377,-82.007,-175.712,8.095,148.335
C00895=1220.968,414.130,-81.972,-175.712,8.092,148.335
C00896=1220.972,413.882,-81.937,-175.713,8.090,148.334
C00897=1220.977,413.634,-81.902,-175.714,8.088,148.334
C00898=1220.981,413.386,-81.867,-175.714,8.086,148.333
C00899=1220.984,413.139,-81.833,-175.714,8.084,148.333
C00900=1220.988,412.892,-81.798,-175.715,8.082,148.332
C00901=1220.992,412.643,-81.763,-175.715,8.080,148.332
C00902=1220.997,412.396,-81.729,-175.716,8.077,148.332
C00903=1221.000,412.149,-81.693,-175.717,8.075,148.331
C00904=1221.004,411.901,-81.659,-175.717,8.073,148.331
C00905=1221.009,411.654,-81.625,-175.717,8.071,148.330
C00906=1221.013,411.406,-81.590,-175.718,8.069,148.330
C00907=1221.017,411.159,-81.555,-175.718,8.066,148.329
C00908=1221.021,410.911,-81.520,-175.719,8.064,148.329
C00909=1221.025,410.664,-81.486,-175.720,8.062,148.329
C00910=1221.029,410.416,-81.451,-175.720,8.059,148.328
C00911=1221.033,410.169,-81.416,-175.721,8.057,148.328
C00912=1221.037,409.921,-81.381,-175.721,8.055,148.327
C00913=1221.041,409.674,-81.347,-175.722,8.053,148.327
C00914=1221.045,409.426,-81.313,-175.722,8.051,148.326
C00915=1221.049,409.178,-81.278,-175.723,8.049,148.326
C00916=1221.053,408.931,-81.243,-175.724,8.046,148.326
C00917=1221.057,408.684,-81.209,-175.724,8.044,148.325
C00918=1221.061,408.435,-81.174,-175.725,8.042,148.325
C00919=1221.065,408.188,-81.139,-175.725,8.040,148.324
C00920=1221.069,407.940,-81.105,-175.725,8.038,148.324
C00921=1221.073,407.693,-81.071,-175.726,8.034,148.323
C00922=1221.077,407.445,-81.035,-175.727,8.032,148.323
C00923=1221.081,407.198,-81.001,-175.727,8.030,148.322
C00924=1221.086,406.950,-80.966,-175.728,8.028,148.322
C00925=1221.089,406.703,-80.932,-175.728,8.026,148.322
C00926=1221.094,406.455,-80.898,-175.729,8.023,148.321
C00927=1221.098,406.207,-80.863,-175.730,8.021,148.321
C00928=1221.102,405.960,-80.829,-175.730,8.019,148.320
C00929=1221.106,405.712,-80.794,-175.731,8.017,148.320
C00930=1221.110,405.464,-80.760,-175.731,8.014,148.319
C00931=1221.113,405.217,-80.725,-175.732,8.012,148.319
C00932=1221.118,404.970,-80.690,-175.733,8.010,148.319
C00933=1221.122,404.722,-80.656,-175.733,8.008,148.318
C00934=1221.126,404.474,-80.621,-175.734,8.005,148.318
C00935=1221.130,404.227,-80.587,-175.734,8.002,148.317
C00936=1221.134,403.979,-80.552,-175.735,8.001,148.317
C00937=1221.139,403.732,-80.518,-175.736,7.997,148.316
C00938=1221.142,403.484,-80.483,-175.736,7.995,148.316
C00939=1221.146,403.236,-80.449,-175.737,7.993,148.316
C00940=1221.151,402.989,-80.414,-175.737,7.991,148.315
C00941=1221.154,402.741,-80.380,-175.738,7.988,148.315
C00942=1221.159,402.494,-80.346,-175.738,7.986,148.314
C00943=1221.162,402.246,-80.312,-175.739,7.984,148.314
C00944=1221.167,401.999,-80.277,-175.740,7.981,148.313
C00945=1221.171,401.751,-80.243,-175.740,7.979,148.313
C00946=1221.174,401.503,-80.208,-175.741,7.977,148.312
C00947=1221.179,401.256,-80.174,-175.742,7.974,148.312
C00948=1221.183,401.008,-80.139,-175.742,7.972,148.312
C00949=1221.187,400.761,-80.105,-175.743,7.970,148.311
C00950=1221.191,400.513,-80.071,-175.744,7.967,148.311
C00951=1221.195,400.265,-80.036,-175.744,7.965,148.310
C00952=1221.199,400.018,-80.002,-175.745,7.963,148.310
C00953=1221.203,399.770,-79.967,-175.746,7.960,148.309
C00954=1221.207,399.523,-79.933,-175.746,7.958,148.309
C00955=1221.211,399.275,-79.899,-175.747,7.955,148.308
C00956=1221.215,399.027,-79.864,-175.748,7.953,148.308
C00957=1221.219,398.780,-79.830,-175.748,7.950,148.307
C00958=1221.223,398.532,-79.795,-175.749,7.948,148.307
C00959=1221.227,398.285,-79.761,-175.749,7.945,148.307
C00960=1221.232,398.037,-79.728,-175.751,7.943,148.306
C00961=1221.236,397.789,-79.693,-175.751,7.941,148.306
C00962=1221.240,397.542,-79.659,-175.751,7.938,148.305
C00963=1221.244,397.294,-79.625,-175.753,7.935,148.305
C00964=1221.248,397.046,-79.590,-175.753,7.934,148.305
C00965=1221.252,396.799,-79.556,-175.754,7.930,148.304
C00966=1221.256,396.552,-79.522,-175.755,7.928,148.304
C00967=1221.260,396.304,-79.487,-175.755,7.925,148.303
C00968=1221.264,396.056,-79.454,-175.756,7.923,148.303
C00969=1221.269,395.809,-79.420,-175.757,7.921,148.302
C00970=1221.273,395.560,-79.385,-175.757,7.918,148.302
C00971=1221.276,395.313,-79.351,-175.758,7.916,148.301
C00972=1221.281,395.066,-79.316,-175.759,7.913,148.301
C00973=1221.284,394.818,-79.282,-175.759,7.911,148.300
C00974=1221.289,394.570,-79.248,-175.761,7.908,148.300
C00975=1221.293,394.323,-79.214,-175.761,7.906,148.300
C00976=1221.297,394.075,-79.180,-175.762,7.903,148.299
C00977=1221.301,393.828,-79.146,-175.763,7.901,148.299
C00978=1221.305,393.580,-79.111,-175.763,7.898,148.298
C00979=1221.310,393.298,-79.073,-175.764,7.895,148.298
C00980=1221.315,393.017,-79.034,-175.765,7.892,148.297
C00981=1221.319,392.735,-78.996,-175.766,7.889,148.297
C00982=1221.323,392.453,-78.957,-175.767,7.886,148.296
C00983=1221.327,392.205,-78.923,-175.768,7.884,148.296
C00984=1221.331,391.958,-78.889,-175.769,7.882,148.295
C00985=1221.336,391.710,-78.854,-175.769,7.879,148.295
C00986=1221.339,391.462,-78.820,-175.770,7.876,148.294
C00987=1221.344,391.214,-78.786,-175.771,7.874,148.294
C00988=1221.348,390.967,-78.752,-175.772,7.872,148.294
C00989=1221.352,390.719,-78.718,-175.773,7.869,148.293
C00990=1221.356,390.472,-78.684,-175.773,7.867,148.293
C00991=1221.360,390.224,-78.650,-175.775,7.864,148.292
C00992=1221.364,389.977,-78.616,-175.775,7.861,148.292
C00993=1221.368,389.729,-78.582,-175.776,7.859,148.291
C00994=1221.372,389.481,-78.548,-175.777,7.856,148.291
C00995=1221.376,389.234,-78.514,-175.778,7.854,148.291
C00996=1221.380,388.986,-78.479,-175.779,7.851,148.290
C00997=1221.384,388.738,-78.446,-175.779,7.849,148.290
C00998=1221.389,388.491,-78.412,-175.780,7.846,148.289
C00999=1221.393,388.243,-78.379,-175.782,7.843,148.289
C01000=1221.396,387.995,-78.344,-175.782,7.841,148.288
C01001=1221.401,387.748,-78.310,-175.783,7.838,148.288
C01002=1221.405,387.500,-78.277,-175.784,7.835,148.288
C01003=1221.410,387.253,-78.242,-175.785,7.833,148.287
C01004=1221.413,387.004,-78.209,-175.785,7.830,148.287
C01005=1221.417,386.757,-78.175,-175.787,7.827,148.286
C01006=1221.422,386.510,-78.140,-175.787,7.825,148.286
C01007=1221.426,386.262,-78.107,-175.788,7.822,148.286
C01008=1221.429,386.014,-78.073,-175.790,7.820,148.285
C01009=1221.434,385.766,-78.039,-175.790,7.817,148.285
C01010=1221.438,385.519,-78.005,-175.791,7.815,148.284
C01011=1221.442,385.271,-77.972,-175.792,7.812,148.284
C01012=1221.446,385.023,-77.937,-175.793,7.809,148.283
C01013=1221.450,384.775,-77.904,-175.794,7.807,148.283
C01014=1221.454,384.528,-77.870,-175.795,7.804,148.283
C01015=1221.459,384.280,-77.837,-175.796,7.801,148.282
C01016=1221.462,384.033,-77.803,-175.797,7.798,148.282
C01017=1221.466,383.785,-77.769,-175.798,7.796,148.281
C01018=1221.470,383.537,-77.735,-175.799,7.793,148.281
C01019=1221.475,383.289,-77.702,-175.800,7.791,148.281
C01020=1221.478,383.042,-77.668,-175.801,7.788,148.280
C01021=1221.483,382.794,-77.634,-175.802,7.785,148.280
C01022=1221.487,382.547,-77.600,-175.803,7.783,148.279
C01023=1221.491,382.299,-77.567,-175.804,7.780,148.279
C01024=1221.495,382.052,-77.533,-175.805,7.777,148.278
C01025=1221.499,381.804,-77.499,-175.806,7.774,148.278
C01026=1221.504,381.556,-77.466,-175.807,7.771,148.278
C01027=1221.507,381.308,-77.432,-175.808,7.769,148.277
C01028=1221.512,381.060,-77.398,-175.809,7.767,148.277
C01029=1221.515,380.813,-77.364,-175.810,7.764,148.277
C01030=1221.520,380.565,-77.331,-175.812,7.761,148.276
C01031=1221.524,380.317,-77.298,-175.813,7.758,148.276
C01032=1221.528,380.069,-77.263,-175.814,7.755,148.275
C01033=1221.532,379.822,-77.230,-175.814,7.753,148.275
C01034=1221.536,379.574,-77.197,-175.815,7.750,148.274
C01035=1221.540,379.327,-77.163,-175.816,7.747,148.274
C01036=1221.545,379.079,-77.129,-175.818,7.745,148.274
C01037=1221.549,378.831,-77.096,-175.819,7.742,148.273
C01038=1221.552,378.583,-77.061,-175.820,7.739,148.273
C01039=1221.556,378.335,-77.028,-175.821,7.736,148.272
C01040=1221.560,378.088,-76.995,-175.822,7.734,148.272
C01041=1221.565,377.840,-76.961,-175.823,7.731,148.272
C01042=1221.569,377.593,-76.928,-175.824,7.729,148.271
C01043=1221.573,377.345,-76.894,-175.825,7.726,148.271
C01044=1221.577,377.098,-76.861,-175.827,7.723,148.270
C01045=1221.581,376.850,-76.827,-175.828,7.720,148.270
C01046=1221.585,376.602,-76.794,-175.829,7.718,148.270
C01047=1221.590,376.354,-76.760,-175.831,7.715,148.270
C01048=1221.593,376.106,-76.726,-175.832,7.712,148.269
C01049=1221.598,375.859,-76.693,-175.833,7.709,148.269
C01050=1221.602,375.611,-76.660,-175.834,7.706,148.268
C01051=1221.606,375.363,-76.627,-175.835,7.703,148.268
C01052=1221.610,375.116,-76.594,-175.836,7.701,148.268
C01053=1221.614,374.868,-76.560,-175.838,7.698,148.267
C01054=1221.617,374.620,-76.526,-175.839,7.695,148.267
C01055=1221.622,374.372,-76.492,-175.840,7.692,148.266
C01056=1221.626,374.124,-76.459,-175.842,7.690,148.266
C01057=1221.630,373.877,-76.426,-175.843,7.687,148.266
C01058=1221.635,373.629,-76.393,-175.844,7.684,148.265
C01059=1221.638,373.382,-76.359,-175.845,7.681,148.265
C01060=1221.643,373.134,-76.326,-175.846,7.678,148.265
C01061=1221.647,372.886,-76.293,-175.847,7.676,148.264
C01062=1221.651,372.638,-76.260,-175.849,7.673,148.264
C01063=1221.655,372.391,-76.227,-175.850,7.670,148.264
C01064=1221.659,372.143,-76.193,-175.851,7.667,148.263
C01065=1221.663,371.895,-76.160,-175.853,7.665,148.263
C01066=1221.667,371.647,-76.127,-175.854,7.662,148.262
C01067=1221.672,371.399,-76.093,-175.855,7.659,148.262
C01068=1221.676,371.151,-76.060,-175.857,7.656,148.262
C01069=1221.680,370.903,-76.027,-175.858,7.654,148.261
C01070=1221.684,370.656,-75.993,-175.859,7.651,148.261
C01071=1221.688,370.408,-75.960,-175.861,7.648,148.261
C01072=1221.692,370.160,-75.927,-175.862,7.645,148.260
C01073=1221.697,369.912,-75.894,-175.863,7.643,148.260
C01074=1221.701,369.665,-75.861,-175.864,7.640,148.260
C01075=1221.705,369.417,-75.828,-175.866,7.637,148.259
C01076=1221.709,369.169,-75.795,-175.867,7.634,148.259
C01077=1221.713,368.922,-75.761,-175.868,7.632,148.259
C01078=1221.717,368.674,-75.728,-175.870,7.629,148.258
C01079=1221.721,368.426,-75.695,-175.872,7.625,148.258
C01080=1221.725,368.178,-75.662,-175.873,7.623,148.258
C01081=1221.730,367.931,-75.629,-175.874,7.620,148.257
C01082=1221.734,367.683,-75.596,-175.876,7.617,148.257
C01083=1221.738,367.403,-75.558,-175.877,7.614,148.257
C01084=1221.743,367.123,-75.521,-175.879,7.611,148.256
C01085=1221.748,366.844,-75.484,-175.881,7.607,148.256
C01086=1221.752,366.564,-75.446,-175.882,7.605,148.256
C01087=1221.756,366.317,-75.414,-175.883,7.602,148.255
C01088=1221.760,366.069,-75.380,-175.885,7.599,148.255
C01089=1221.764,365.820,-75.348,-175.886,7.596,148.255
C01090=1221.769,365.573,-75.315,-175.888,7.593,148.254
C01091=1221.773,365.325,-75.282,-175.889,7.590,148.254
C01092=1221.777,365.077,-75.249,-175.891,7.588,148.254
C01093=1221.781,364.830,-75.215,-175.892,7.585,148.253
C01094=1221.785,364.582,-75.182,-175.894,7.582,148.253
C01095=1221.790,364.333,-75.150,-175.895,7.580,148.253
C01096=1221.793,364.086,-75.117,-175.897,7.576,148.253
C01097=1221.797,363.838,-75.084,-175.898,7.573,148.252
C01098=1221.801,363.591,-75.051,-175.900,7.571,148.252
C01099=1221.806,363.342,-75.018,-175.901,7.568,148.252
C01100=1221.810,363.094,-74.985,-175.903,7.566,148.251
C01101=1221.814,362.847,-74.952,-175.904,7.562,148.251
C01102=1221.817,362.599,-74.920,-175.906,7.559,148.251
C01103=1221.822,362.351,-74.887,-175.907,7.557,148.250
C01104=1221.826,362.103,-74.854,-175.909,7.554,148.250
C01105=1221.830,361.856,-74.821,-175.910,7.551,148.250
C01106=1221.835,361.607,-74.788,-175.912,7.548,148.250
C01107=1221.839,361.360,-74.756,-175.914,7.545,148.249
C01108=1221.843,361.113,-74.723,-175.915,7.542,148.249
C01109=1221.847,360.864,-74.691,-175.917,7.540,148.249
C01110=1221.851,360.617,-74.657,-175.918,7.536,148.248
C01111=1221.855,360.369,-74.624,-175.920,7.534,148.248
C01112=1221.859,360.121,-74.592,-175.922,7.531,148.248
C01113=1221.863,359.873,-74.559,-175.923,7.528,148.248
C01114=1221.867,359.625,-74.526,-175.925,7.525,148.247
C01115=1221.872,359.377,-74.494,-175.927,7.523,148.247
C01116=1221.875,359.130,-74.461,-175.928,7.520,148.247
C01117=1221.880,358.882,-74.429,-175.929,7.517,148.247
C01118=1221.884,358.634,-74.396,-175.932,7.514,148.246
C01119=1221.889,358.387,-74.363,-175.933,7.511,148.246
C01120=1221.892,358.139,-74.331,-175.934,7.508,148.246
C01121=1221.896,357.891,-74.298,-175.936,7.506,148.246
C01122=1221.901,357.642,-74.265,-175.938,7.502,148.245
C01123=1221.904,357.395,-74.233,-175.939,7.500,148.245
C01124=1221.909,357.147,-74.201,-175.941,7.497,148.245
C01125=1221.913,356.900,-74.168,-175.943,7.495,148.245
C01126=1221.917,356.652,-74.136,-175.944,7.491,148.244
C01127=1221.921,356.404,-74.103,-175.946,7.489,148.244
C01128=1221.926,356.156,-74.070,-175.948,7.486,148.244
C01129=1221.929,355.908,-74.038,-175.949,7.483,148.244
C01130=1221.934,355.660,-74.005,-175.951,7.480,148.243
C01131=1221.939,355.412,-73.973,-175.953,7.477,148.243
C01132=1221.942,355.165,-73.940,-175.954,7.475,148.243
C01133=1221.946,354.916,-73.908,-175.956,7.471,148.243
C01134=1221.951,354.669,-73.875,-175.958,7.469,148.242
C01135=1221.954,354.421,-73.843,-175.960,7.466,148.242
C01136=1221.959,354.173,-73.811,-175.961,7.464,148.242
C01137=1221.963,353.925,-73.778,-175.963,7.460,148.242
C01138=1221.967,353.677,-73.746,-175.965,7.458,148.241
C01139=1221.972,353.429,-73.714,-175.966,7.455,148.241
C01140=1221.975,353.181,-73.681,-175.969,7.452,148.241
C01141=1221.980,352.934,-73.649,-175.970,7.449,148.241
C01142=1221.984,352.686,-73.617,-175.971,7.446,148.240
C01143=1221.988,352.438,-73.584,-175.974,7.443,148.240
C01144=1221.992,352.190,-73.551,-175.975,7.441,148.240
C01145=1221.997,351.942,-73.520,-175.977,7.438,148.240
C01146=1222.001,351.695,-73.487,-175.978,7.435,148.240
C01147=1222.005,351.447,-73.455,-175.981,7.432,148.239
C01148=1222.009,351.198,-73.423,-175.982,7.430,148.239
C01149=1222.013,350.951,-73.391,-175.984,7.427,148.239
C01150=1222.017,350.703,-73.358,-175.986,7.424,148.239
C01151=1222.021,350.455,-73.326,-175.988,7.421,148.239
C01152=1222.026,350.207,-73.294,-175.989,7.419,148.238
C01153=1222.030,349.959,-73.262,-175.992,7.415,148.238
C01154=1222.034,349.711,-73.230,-175.993,7.413,148.238
C01155=1222.038,349.464,-73.197,-175.995,7.410,148.238
C01156=1222.042,349.215,-73.165,-175.997,7.407,148.238
C01157=1222.046,348.968,-73.133,-175.999,7.404,148.237
C01158=1222.051,348.720,-73.101,-176.000,7.402,148.237
C01159=1222.055,348.472,-73.069,-176.002,7.398,148.237
C01160=1222.060,348.224,-73.037,-176.004,7.396,148.237
C01161=1222.063,347.976,-73.005,-176.006,7.393,148.237
C01162=1222.067,347.728,-72.972,-176.008,7.390,148.236
C01163=1222.071,347.480,-72.940,-176.010,7.388,148.236
C01164=1222.076,347.233,-72.909,-176.011,7.385,148.236
C01165=1222.080,346.984,-72.876,-176.013,7.382,148.236
C01166=1222.084,346.736,-72.844,-176.015,7.379,148.236
C01167=1222.089,346.489,-72.812,-176.017,7.377,148.235
C01168=1222.092,346.241,-72.780,-176.019,7.373,148.235
C01169=1222.096,345.993,-72.748,-176.020,7.371,148.235
C01170=1222.101,345.745,-72.716,-176.022,7.368,148.235
C01171=1222.105,345.497,-72.685,-176.024,7.365,148.235
C01172=1222.109,345.249,-72.652,-176.026,7.362,148.234
C01173=1222.114,345.001,-72.621,-176.028,7.360,148.234
C01174=1222.117,344.753,-72.589,-176.030,7.357,148.234
C01175=1222.122,344.505,-72.556,-176.032,7.354,148.234
C01176=1222.126,344.258,-72.525,-176.033,7.352,148.234
C01177=1222.130,344.009,-72.493,-176.036,7.348,148.234
C01178=1222.135,343.762,-72.461,-176.037,7.346,148.233
C01179=1222.139,343.514,-72.429,-176.039,7.343,148.233
C01180=1222.142,343.266,-72.397,-176.041,7.340,148.233
C01181=1222.148,343.017,-72.366,-176.043,7.338,148.233
C01182=1222.151,342.769,-72.334,-176.045,7.334,148.233
C01183=1222.155,342.521,-72.302,-176.047,7.332,148.233
C01184=1222.160,342.274,-72.270,-176.049,7.329,148.233
C01185=1222.164,342.026,-72.238,-176.051,7.326,148.232
C01186=1222.168,341.778,-72.207,-176.053,7.324,148.232
C01187=1222.173,341.500,-72.171,-176.055,7.320,148.232
C01188=1222.178,341.222,-72.136,-176.057,7.317,148.232
C01189=1222.182,340.945,-72.100,-176.059,7.314,148.232
C01190=1222.187,340.667,-72.065,-176.061,7.311,148.231
C01191=1222.191,340.418,-72.033,-176.063,7.309,148.232
C01192=1222.195,340.171,-72.001,-176.065,7.306,148.231
C01193=1222.199,339.923,-71.969,-176.067,7.303,148.231
C01194=1222.203,339.676,-71.938,-176.070,7.300,148.231
C01195=1222.208,339.427,-71.906,-176.071,7.297,148.231
C01196=1222.213,339.179,-71.875,-176.073,7.295,148.231
C01197=1222.216,338.931,-71.843,-176.075,7.292,148.230
C01198=1222.220,338.683,-71.812,-176.077,7.289,148.231
C01199=1222.225,338.435,-71.780,-176.079,7.287,148.230
C01200=1222.228,338.187,-71.748,-176.081,7.283,148.230
C01201=1222.233,337.940,-71.716,-176.083,7.281,148.230
C01202=1222.237,337.691,-71.685,-176.085,7.278,148.230
C01203=1222.242,337.444,-71.654,-176.087,7.275,148.230
C01204=1222.246,337.195,-71.623,-176.089,7.273,148.230
C01205=1222.250,336.948,-71.591,-176.091,7.270,148.230
C01206=1222.254,336.700,-71.559,-176.093,7.267,148.229
C01207=1222.258,336.452,-71.529,-176.095,7.265,148.229
C01208=1222.263,336.203,-71.496,-176.097,7.262,148.229
C01209=1222.267,335.956,-71.465,-176.099,7.259,148.229
C01210=1222.271,335.707,-71.433,-176.102,7.256,148.229
C01211=1222.275,335.460,-71.402,-176.103,7.254,148.229
C01212=1222.279,335.211,-71.371,-176.105,7.251,148.229
C01213=1222.284,334.964,-71.339,-176.107,7.248,148.229
C01214=1222.288,334.715,-71.308,-176.109,7.245,148.228
C01215=1222.292,334.468,-71.277,-176.112,7.242,148.228
C01216=1222.296,334.219,-71.246,-176.113,7.240,148.228
C01217=1222.300,333.972,-71.214,-176.115,7.237,148.228
C01218=1222.304,333.723,-71.183,-176.118,7.234,148.228
C01219=1222.309,333.476,-71.152,-176.119,7.232,148.228
C01220=1222.313,333.227,-71.120,-176.122,7.229,148.228
C01221=1222.317,332.980,-71.089,-176.124,7.226,148.228
C01222=1222.321,332.731,-71.058,-176.126,7.224,148.228
C01223=1222.325,332.484,-71.026,-176.128,7.221,148.228
C01224=1222.330,332.236,-70.996,-176.129,7.218,148.227
C01225=1222.334,331.987,-70.964,-176.132,7.216,148.227
C01226=1222.338,331.740,-70.933,-176.134,7.212,148.227
C01227=1222.342,331.491,-70.902,-176.136,7.210,148.227
C01228=1222.346,331.244,-70.870,-176.138,7.207,148.227
C01229=1222.351,330.995,-70.839,-176.140,7.205,148.227
C01230=1222.355,330.747,-70.808,-176.142,7.202,148.227
C01231=1222.359,330.500,-70.777,-176.144,7.199,148.227
C01232=1222.363,330.251,-70.746,-176.146,7.197,148.227
C01233=1222.368,330.003,-70.715,-176.149,7.194,148.227
C01234=1222.372,329.755,-70.683,-176.150,7.191,148.227
C01235=1222.376,329.507,-70.653,-176.152,7.189,148.227
C01236=1222.381,329.259,-70.622,-176.155,7.185,148.226
C01237=1222.385,329.011,-70.591,-176.157,7.183,148.226
C01238=1222.389,328.763,-70.559,-176.159,7.180,148.226
C01239=1222.393,328.515,-70.528,-176.161,7.178,148.226
C01240=1222.398,328.267,-70.497,-176.163,7.175,148.226
C01241=1222.402,328.019,-70.467,-176.165,7.172,148.226
C01242=1222.406,327.771,-70.435,-176.167,7.170,148.226
C01243=1222.410,327.523,-70.404,-176.170,7.166,148.226
C01244=1222.415,327.275,-70.374,-176.172,7.164,148.226
C01245=1222.419,327.027,-70.343,-176.173,7.162,148.226
C01246=1222.423,326.779,-70.312,-176.176,7.159,148.226
C01247=1222.427,326.532,-70.281,-176.178,7.156,148.226
C01248=1222.431,326.283,-70.250,-176.180,7.153,148.226
C01249=1222.436,326.035,-70.219,-176.182,7.151,148.226
C01250=1222.440,325.786,-70.188,-176.184,7.148,148.225
C01251=1222.444,325.538,-70.157,-176.187,7.145,148.225
C01252=1222.449,325.290,-70.126,-176.189,7.143,148.225
C01253=1222.453,325.043,-70.096,-176.191,7.140,148.225
C01254=1222.457,324.794,-70.065,-176.193,7.137,148.225
C01255=1222.461,324.546,-70.034,-176.195,7.135,148.225
C01256=1222.466,324.299,-70.003,-176.197,7.132,148.225
C01257=1222.469,324.050,-69.972,-176.200,7.130,148.225
C01258=1222.473,323.803,-69.942,-176.202,7.127,148.225
C01259=1222.478,323.555,-69.911,-176.204,7.124,148.225
C01260=1222.482,323.306,-69.880,-176.206,7.122,148.225
C01261=1222.486,323.058,-69.849,-176.209,7.119,148.225
C01262=1222.491,322.810,-69.819,-176.210,7.116,148.225
C01263=1222.495,322.562,-69.788,-176.213,7.113,148.225
C01264=1222.498,322.314,-69.757,-176.215,7.111,148.225
C01265=1222.503,322.066,-69.727,-176.217,7.109,148.225
C01266=1222.508,321.818,-69.696,-176.219,7.105,148.225
C01267=1222.511,321.569,-69.666,-176.221,7.103,148.225
C01268=1222.516,321.321,-69.635,-176.224,7.100,148.225
C01269=1222.521,321.073,-69.605,-176.226,7.098,148.225
C01270=1222.524,320.826,-69.574,-176.228,7.095,148.225
C01271=1222.528,320.577,-69.543,-176.230,7.092,148.225
C01272=1222.533,320.329,-69.512,-176.232,7.090,148.224
C01273=1222.537,320.081,-69.482,-176.235,7.087,148.224
C01274=1222.542,319.833,-69.452,-176.237,7.085,148.224
C01275=1222.546,319.585,-69.421,-176.239,7.082,148.225
C01276=1222.550,319.336,-69.391,-176.241,7.079,148.224
C01277=1222.554,319.088,-69.360,-176.243,7.077,148.224
C01278=1222.559,318.840,-69.329,-176.245,7.075,148.224
C01279=1222.563,318.593,-69.299,-176.248,7.072,148.224
C01280=1222.567,318.344,-69.268,-176.250,7.069,148.224
C01281=1222.571,318.096,-69.239,-176.252,7.066,148.224
C01282=1222.576,317.848,-69.208,-176.254,7.064,148.224
C01283=1222.579,317.600,-69.178,-176.257,7.062,148.224
C01284=1222.584,317.352,-69.147,-176.259,7.058,148.224
C01285=1222.589,317.104,-69.117,-176.261,7.056,148.224
C01286=1222.592,316.855,-69.086,-176.263,7.053,148.224
C01287=1222.597,316.607,-69.056,-176.266,7.051,148.224
C01288=1222.601,316.359,-69.026,-176.268,7.048,148.224
C01289=1222.606,316.111,-68.995,-176.270,7.045,148.224
C01290=1222.610,315.864,-68.965,-176.272,7.043,148.224
C01291=1222.615,315.587,-68.932,-176.275,7.040,148.224
C01292=1222.619,315.312,-68.898,-176.277,7.037,148.224
C01293=1222.624,315.035,-68.864,-176.280,7.034,148.224
C01294=1222.629,314.759,-68.830,-176.282,7.031,148.224
C01295=1222.633,314.511,-68.801,-176.285,7.028,148.224
C01296=1222.637,314.263,-68.770,-176.287,7.026,148.224
C01297=1222.641,314.016,-68.740,-176.289,7.024,148.224
C01298=1222.646,313.767,-68.710,-176.292,7.021,148.224
C01299=1222.650,313.519,-68.680,-176.294,7.019,148.224
C01300=1222.654,313.271,-68.650,-176.296,7.016,148.224
C01301=1222.659,313.023,-68.619,-176.298,7.013,148.224
C01302=1222.662,312.774,-68.590,-176.300,7.011,148.224
C01303=1222.667,312.526,-68.559,-176.303,7.008,148.224
C01304=1222.671,312.278,-68.529,-176.305,7.006,148.224
C01305=1222.675,312.030,-68.499,-176.308,7.003,148.224
C01306=1222.680,311.782,-68.469,-176.310,7.000,148.224
C01307=1222.684,311.534,-68.439,-176.312,6.998,148.224
C01308=1222.689,311.286,-68.409,-176.314,6.995,148.224
C01309=1222.693,311.038,-68.379,-176.317,6.993,148.224
C01310=1222.697,310.790,-68.349,-176.319,6.991,148.224
C01311=1222.701,310.542,-68.318,-176.321,6.988,148.224
C01312=1222.706,310.293,-68.289,-176.323,6.985,148.224
C01313=1222.710,310.045,-68.260,-176.326,6.982,148.224
C01314=1222.714,309.797,-68.229,-176.328,6.980,148.224
C01315=1222.719,309.549,-68.199,-176.330,6.978,148.224
C01316=1222.723,309.301,-68.170,-176.332,6.975,148.224
C01317=1222.727,309.053,-68.139,-176.335,6.972,148.224
C01318=1222.731,308.804,-68.109,-176.337,6.970,148.224
C01319=1222.735,308.556,-68.079,-176.339,6.967,148.224
C01320=1222.740,308.307,-68.049,-176.341,6.965,148.225
C01321=1222.744,308.059,-68.020,-176.344,6.962,148.225
C01322=1222.748,307.811,-67.990,-176.346,6.960,148.225
C01323=1222.753,307.563,-67.959,-176.348,6.957,148.225
C01324=1222.757,307.315,-67.930,-176.351,6.954,148.225
C01325=1222.761,307.066,-67.901,-176.353,6.952,148.225
C01326=1222.765,306.818,-67.871,-176.355,6.950,148.225
C01327=1222.770,306.570,-67.840,-176.358,6.947,148.225
C01328=1222.774,306.322,-67.811,-176.360,6.945,148.225
C01329=1222.779,306.074,-67.782,-176.363,6.942,148.225
C01330=1222.783,305.826,-67.752,-176.365,6.939,148.225
C01331=1222.787,305.578,-67.722,-176.367,6.937,148.225
C01332=1222.792,305.330,-67.692,-176.370,6.934,148.225
C01333=1222.796,305.082,-67.663,-176.372,6.932,148.225
C01334=1222.800,304.833,-67.633,-176.374,6.930,148.225
C01335=1222.804,304.585,-67.604,-176.376,6.927,148.225
C01336=1222.809,304.337,-67.574,-176.379,6.924,148.225
C01337=1222.814,304.088,-67.544,-176.381,6.922,148.225
C01338=1222.817,303.841,-67.514,-176.384,6.919,148.225
C01339=1222.822,303.592,-67.485,-176.386,6.917,148.225
C01340=1222.826,303.344,-67.455,-176.389,6.914,148.225
C01341=1222.830,303.096,-67.426,-176.391,6.912,148.226
C01342=1222.834,302.848,-67.396,-176.393,6.910,148.226
C01343=1222.838,302.599,-67.367,-176.395,6.907,148.226
C01344=1222.843,302.351,-67.337,-176.398,6.905,148.226
C01345=1222.848,302.103,-67.308,-176.400,6.902,148.226
C01346=1222.852,301.855,-67.278,-176.402,6.899,148.226
C01347=1222.856,301.607,-67.249,-176.404,6.897,148.226
C01348=1222.861,301.358,-67.219,-176.407,6.895,148.226
C01349=1222.865,301.110,-67.190,-176.409,6.892,148.226
C01350=1222.869,300.862,-67.160,-176.412,6.890,148.226
C01351=1222.873,300.614,-67.131,-176.414,6.888,148.226
C01352=1222.877,300.365,-67.101,-176.417,6.885,148.226
C01353=1222.881,300.117,-67.072,-176.419,6.882,148.226
C01354=1222.886,299.869,-67.043,-176.421,6.880,148.226
C01355=1222.890,299.621,-67.013,-176.423,6.877,148.226
C01356=1222.895,299.373,-66.984,-176.426,6.875,148.226
C01357=1222.899,299.124,-66.955,-176.428,6.873,148.226
C01358=1222.903,298.876,-66.926,-176.431,6.870,148.227
C01359=1222.907,298.627,-66.896,-176.433,6.868,148.227
C01360=1222.912,298.379,-66.867,-176.436,6.865,148.227
C01361=1222.916,298.132,-66.838,-176.438,6.863,148.227
C01362=1222.921,297.883,-66.808,-176.440,6.860,148.227
C01363=1222.925,297.635,-66.779,-176.443,6.857,148.227
C01364=1222.929,297.386,-66.750,-176.445,6.855,148.227
C01365=1222.933,297.138,-66.721,-176.447,6.853,148.227
C01366=1222.938,296.890,-66.691,-176.450,6.850,148.227
C01367=1222.942,296.642,-66.662,-176.452,6.848,148.227
C01368=1222.947,296.393,-66.633,-176.454,6.846,148.227
C01369=1222.951,296.145,-66.604,-176.457,6.843,148.227
C01370=1222.955,295.897,-66.575,-176.459,6.841,148.228
C01371=1222.959,295.648,-66.545,-176.461,6.839,148.228
C01372=1222.965,295.400,-66.517,-176.464,6.835,148.228
C01373=1222.968,295.152,-66.488,-176.466,6.833,148.228
C01374=1222.972,294.904,-66.458,-176.468,6.831,148.228
C01375=1222.977,294.655,-66.430,-176.471,6.829,148.228
C01376=1222.981,294.408,-66.401,-176.474,6.826,148.228
C01377=1222.986,294.159,-66.371,-176.476,6.824,148.228
C01378=1222.990,293.910,-66.342,-176.478,6.822,148.228
C01379=1222.994,293.662,-66.313,-176.481,6.819,148.228
C01380=1222.998,293.415,-66.284,-176.483,6.817,148.229
C01381=1223.003,293.166,-66.256,-176.485,6.815,148.229
C01382=1223.007,292.918,-66.226,-176.488,6.811,148.229
C01383=1223.011,292.669,-66.197,-176.490,6.809,148.229
C01384=1223.016,292.421,-66.168,-176.493,6.807,148.229
C01385=1223.020,292.173,-66.139,-176.495,6.804,148.229
C01386=1223.024,291.924,-66.111,-176.497,6.802,148.229
C01387=1223.028,291.676,-66.081,-176.500,6.800,148.229
C01388=1223.033,291.428,-66.053,-176.503,6.797,148.229
C01389=1223.038,291.180,-66.024,-176.505,6.795,148.229
C01390=1223.041,290.931,-65.995,-176.507,6.793,148.229
C01391=1223.046,290.684,-65.966,-176.509,6.791,148.230
C01392=1223.051,290.435,-65.938,-176.512,6.788,148.230
C01393=1223.055,290.186,-65.908,-176.514,6.786,148.230
C01394=1223.059,289.938,-65.880,-176.516,6.783,148.230
C01395=1223.064,289.664,-65.849,-176.520,6.781,148.230
C01396=1223.068,289.390,-65.816,-176.522,6.778,148.230
C01397=1223.073,289.116,-65.785,-176.525,6.776,148.230
C01398=1223.078,288.842,-65.753,-176.527,6.773,148.230
C01399=1223.082,288.593,-65.724,-176.530,6.770,148.230
C01400=1223.087,288.345,-65.695,-176.533,6.768,148.231
C01401=1223.091,288.097,-65.667,-176.535,6.765,148.231
C01402=1223.095,287.848,-65.638,-176.537,6.763,148.231
C01403=1223.100,287.600,-65.609,-176.540,6.761,148.231
C01404=1223.104,287.352,-65.581,-176.542,6.758,148.231
C01405=1223.108,287.103,-65.552,-176.544,6.756,148.231
C01406=1223.113,286.855,-65.523,-176.546,6.754,148.231
C01407=1223.117,286.607,-65.495,-176.550,6.751,148.232
C01408=1223.122,286.359,-65.466,-176.552,6.749,148.232
C01409=1223.126,286.110,-65.437,-176.554,6.747,148.232
C01410=1223.130,285.862,-65.409,-176.556,6.745,148.232
C01411=1223.135,285.613,-65.381,-176.559,6.742,148.232
C01412=1223.139,285.365,-65.352,-176.561,6.740,148.232
C01413=1223.144,285.117,-65.324,-176.564,6.738,148.232
C01414=1223.148,284.868,-65.295,-176.566,6.735,148.232
C01415=1223.152,284.620,-65.267,-176.569,6.733,148.233
C01416=1223.157,284.372,-65.238,-176.571,6.731,148.233
C01417=1223.161,284.124,-65.210,-176.573,6.728,148.233
C01418=1223.166,283.875,-65.181,-176.576,6.726,148.233
C01419=1223.169,283.627,-65.153,-176.579,6.723,148.233
C01420=1223.174,283.378,-65.124,-176.581,6.721,148.233
C01421=1223.178,283.130,-65.096,-176.583,6.719,148.233
C01422=1223.182,282.882,-65.067,-176.586,6.716,148.233
C01423=1223.188,282.634,-65.039,-176.588,6.714,148.234
C01424=1223.191,282.385,-65.011,-176.591,6.712,148.234
C01425=1223.196,282.137,-64.982,-176.593,6.710,148.234
C01426=1223.200,281.888,-64.954,-176.596,6.707,148.234
C01427=1223.205,281.640,-64.926,-176.598,6.705,148.234
C01428=1223.209,281.392,-64.897,-176.600,6.703,148.234
C01429=1223.213,281.144,-64.870,-176.603,6.701,148.235
C01430=1223.218,280.895,-64.841,-176.605,6.698,148.235
C01431=1223.222,280.647,-64.813,-176.608,6.696,148.235
C01432=1223.227,280.398,-64.784,-176.610,6.694,148.235
C01433=1223.231,280.150,-64.757,-176.612,6.692,148.235
C01434=1223.235,279.901,-64.728,-176.615,6.689,148.235
C01435=1223.240,279.653,-64.700,-176.618,6.687,148.235
C01436=1223.244,279.405,-64.671,-176.620,6.685,148.236
C01437=1223.249,279.157,-64.644,-176.622,6.683,148.236
C01438=1223.252,278.908,-64.616,-176.625,6.680,148.236
C01439=1223.257,278.660,-64.587,-176.628,6.678,148.236
C01440=1223.261,278.411,-64.559,-176.630,6.675,148.236
C01441=1223.266,278.163,-64.531,-176.632,6.674,148.236
C01442=1223.270,277.915,-64.502,-176.635,6.670,148.236
C01443=1223.274,277.667,-64.475,-176.638,6.669,148.237
C01444=1223.279,277.418,-64.446,-176.640,6.666,148.237
C01445=1223.284,277.169,-64.419,-176.642,6.664,148.237
C01446=1223.287,276.921,-64.391,-176.645,6.661,148.237
C01447=1223.292,276.673,-64.362,-176.647,6.659,148.237
C01448=1223.296,276.424,-64.334,-176.650,6.657,148.237
C01449=1223.301,276.176,-64.306,-176.652,6.655,148.237
C01450=1223.305,275.928,-64.279,-176.654,6.653,148.238
C01451=1223.310,275.679,-64.251,-176.657,6.650,148.238
C01452=1223.314,275.431,-64.223,-176.660,6.648,148.238
C01453=1223.318,275.182,-64.195,-176.662,6.646,148.238
C01454=1223.323,274.934,-64.166,-176.664,6.644,148.238
C01455=1223.327,274.685,-64.139,-176.667,6.641,148.238
C01456=1223.331,274.437,-64.111,-176.670,6.639,148.239
C01457=1223.336,274.189,-64.083,-176.672,6.637,148.239
C01458=1223.340,273.940,-64.055,-176.674,6.635,148.239
C01459=1223.345,273.692,-64.028,-176.676,6.633,148.239
C01460=1223.348,273.443,-63.999,-176.680,6.630,148.239
C01461=1223.353,273.195,-63.972,-176.682,6.628,148.240
C01462=1223.358,272.946,-63.944,-176.684,6.626,148.240
C01463=1223.362,272.698,-63.916,-176.686,6.624,148.240
C01464=1223.366,272.450,-63.888,-176.689,6.622,148.240
C01465=1223.371,272.202,-63.861,-176.692,6.619,148.240
C01466=1223.375,271.953,-63.833,-176.694,6.617,148.241
C01467=1223.380,271.705,-63.805,-176.696,6.615,148.241
C01468=1223.384,271.456,-63.777,-176.699,6.613,148.241
C01469=1223.388,271.208,-63.749,-176.701,6.611,148.241
C01470=1223.393,270.959,-63.722,-176.704,6.608,148.241
C01471=1223.397,270.711,-63.694,-176.706,6.606,148.241
C01472=1223.401,270.463,-63.666,-176.709,6.604,148.242
C01473=1223.406,270.214,-63.639,-176.711,6.602,148.242
C01474=1223.411,269.966,-63.611,-176.714,6.600,148.242
C01475=1223.415,269.717,-63.583,-176.716,6.597,148.242
C01476=1223.419,269.469,-63.556,-176.719,6.595,148.242
C01477=1223.424,269.220,-63.529,-176.721,6.593,148.242
C01478=1223.428,268.972,-63.500,-176.724,6.591,148.243
C01479=1223.432,268.723,-63.473,-176.726,6.589,148.243
C01480=1223.437,268.476,-63.446,-176.729,6.587,148.243
C01481=1223.441,268.226,-63.418,-176.731,6.584,148.243
C01482=1223.446,267.978,-63.390,-176.734,6.582,148.243
C01483=1223.450,267.730,-63.363,-176.736,6.580,148.244
C01484=1223.455,267.481,-63.336,-176.739,6.578,148.244
C01485=1223.459,267.233,-63.308,-176.741,6.576,148.244
C01486=1223.463,266.984,-63.281,-176.743,6.574,148.244
C01487=1223.468,266.736,-63.253,-176.746,6.571,148.244
C01488=1223.472,266.488,-63.226,-176.749,6.569,148.244
C01489=1223.476,266.239,-63.198,-176.751,6.567,148.245
C01490=1223.481,265.991,-63.170,-176.754,6.565,148.245
C01491=1223.485,265.742,-63.143,-176.756,6.563,148.245
C01492=1223.490,265.494,-63.116,-176.758,6.561,148.245
C01493=1223.494,265.245,-63.088,-176.761,6.558,148.245
C01494=1223.499,264.997,-63.061,-176.764,6.556,148.246
C01495=1223.503,264.748,-63.034,-176.766,6.554,148.246
C01496=1223.508,264.500,-63.006,-176.768,6.552,148.246
C01497=1223.512,264.251,-62.979,-176.771,6.550,148.246
C01498=1223.516,264.003,-62.952,-176.773,6.548,148.246
C01499=1223.521,263.730,-62.922,-176.776,6.545,148.247
C01500=1223.526,263.458,-62.892,-176.779,6.543,148.247
C01501=1223.531,263.185,-62.862,-176.782,6.540,148.247
C01502=1223.536,262.912,-62.832,-176.784,6.538,148.247
C01503=1223.539,262.664,-62.805,-176.787,6.536,148.248
C01504=1223.544,262.415,-62.778,-176.789,6.534,148.248
C01505=1223.548,262.167,-62.751,-176.792,6.532,148.248
C01506=1223.553,261.918,-62.724,-176.795,6.530,148.248
C01507=1223.558,261.670,-62.697,-176.797,6.527,148.248
C01508=1223.562,261.422,-62.669,-176.800,6.526,148.249
C01509=1223.566,261.173,-62.641,-176.802,6.523,148.249
C01510=1223.571,260.924,-62.614,-176.804,6.521,148.249
C01511=1223.576,260.676,-62.587,-176.807,6.520,148.249
C01512=1223.579,260.428,-62.561,-176.810,6.517,148.249
C01513=1223.584,260.179,-62.534,-176.812,6.515,148.250
C01514=1223.589,259.931,-62.507,-176.815,6.513,148.250
C01515=1223.593,259.682,-62.480,-176.817,6.511,148.250
C01516=1223.597,259.433,-62.452,-176.819,6.509,148.250
C01517=1223.601,259.185,-62.426,-176.822,6.506,148.250
C01518=1223.606,258.936,-62.399,-176.824,6.505,148.251
C01519=1223.611,258.688,-62.372,-176.827,6.503,148.251
C01520=1223.615,258.439,-62.345,-176.830,6.500,148.251
C01521=1223.620,258.191,-62.318,-176.832,6.498,148.251
C01522=1223.624,257.943,-62.291,-176.835,6.496,148.252
C01523=1223.629,257.694,-62.264,-176.837,6.494,148.252
C01524=1223.633,257.446,-62.237,-176.839,6.492,148.252
C01525=1223.637,257.196,-62.210,-176.842,6.490,148.252
C01526=1223.641,256.948,-62.183,-176.844,6.488,148.253
C01527=1223.646,256.700,-62.156,-176.847,6.486,148.253
C01528=1223.651,256.451,-62.129,-176.849,6.484,148.253
C01529=1223.655,256.203,-62.102,-176.852,6.482,148.253
C01530=1223.659,255.954,-62.075,-176.855,6.479,148.253
C01531=1223.664,255.706,-62.048,-176.857,6.477,148.254
C01532=1223.668,255.457,-62.021,-176.859,6.475,148.254
C01533=1223.672,255.209,-61.995,-176.862,6.473,148.254
C01534=1223.677,254.960,-61.969,-176.865,6.471,148.254
C01535=1223.682,254.712,-61.941,-176.867,6.469,148.255
C01536=1223.686,254.463,-61.915,-176.869,6.467,148.255
C01537=1223.691,254.215,-61.888,-176.872,6.465,148.255
C01538=1223.695,253.966,-61.861,-176.874,6.463,148.255
C01539=1223.699,253.718,-61.834,-176.877,6.461,148.256
C01540=1223.704,253.469,-61.808,-176.879,6.459,148.256
C01541=1223.709,253.221,-61.781,-176.882,6.456,148.256
C01542=1223.713,252.973,-61.755,-176.885,6.454,148.256
C01543=1223.717,252.724,-61.727,-176.887,6.453,148.257
C01544=1223.722,252.475,-61.701,-176.890,6.451,148.257
C01545=1223.726,252.227,-61.675,-176.892,6.448,148.257
C01546=1223.731,251.978,-61.648,-176.895,6.447,148.257
C01547=1223.735,251.730,-61.621,-176.897,6.445,148.258
C01548=1223.740,251.481,-61.595,-176.899,6.443,148.258
C01549=1223.744,251.233,-61.568,-176.902,6.441,148.258
C01550=1223.748,250.984,-61.541,-176.905,6.439,148.258
C01551=1223.753,250.735,-61.515,-176.907,6.437,148.258
C01552=1223.757,250.487,-61.488,-176.909,6.435,148.259
C01553=1223.762,250.238,-61.461,-176.912,6.433,148.259
C01554=1223.766,249.990,-61.436,-176.915,6.430,148.259
C01555=1223.771,249.741,-61.409,-176.917,6.428,148.259
C01556=1223.775,249.492,-61.383,-176.920,6.426,148.260
C01557=1223.780,249.244,-61.356,-176.922,6.424,148.260
C01558=1223.784,248.996,-61.329,-176.925,6.422,148.260
C01559=1223.788,248.747,-61.303,-176.927,6.420,148.260
C01560=1223.792,248.498,-61.276,-176.930,6.418,148.261
C01561=1223.797,248.249,-61.250,-176.932,6.416,148.261
C01562=1223.801,248.001,-61.224,-176.935,6.414,148.261
C01563=1223.806,247.752,-61.197,-176.937,6.412,148.261
C01564=1223.810,247.504,-61.171,-176.940,6.410,148.262
C01565=1223.815,247.255,-61.144,-176.942,6.409,148.262
C01566=1223.820,247.007,-61.118,-176.945,6.406,148.262
C01567=1223.825,246.758,-61.092,-176.947,6.404,148.262
C01568=1223.829,246.510,-61.066,-176.950,6.403,148.263
C01569=1223.833,246.261,-61.040,-176.952,6.401,148.263
C01570=1223.837,246.013,-61.013,-176.955,6.398,148.263
C01571=1223.842,245.764,-60.987,-176.957,6.397,148.263
C01572=1223.846,245.515,-60.960,-176.960,6.395,148.264
C01573=1223.851,245.266,-60.934,-176.962,6.393,148.264
C01574=1223.854,245.018,-60.908,-176.965,6.391,148.264
C01575=1223.860,244.770,-60.882,-176.967,6.389,148.264
C01576=1223.864,244.521,-60.856,-176.970,6.386,148.265
C01577=1223.869,244.273,-60.829,-176.973,6.384,148.265
C01578=1223.873,244.024,-60.803,-176.976,6.382,148.265
C01579=1223.877,243.775,-60.777,-176.978,6.380,148.265
C01580=1223.882,243.526,-60.750,-176.980,6.378,148.266
C01581=1223.886,243.278,-60.725,-176.983,6.376,148.266
C01582=1223.891,243.030,-60.699,-176.986,6.375,148.266
C01583=1223.896,242.781,-60.672,-176.988,6.372,148.266
C01584=1223.900,242.532,-60.646,-176.990,6.370,148.267
C01585=1223.904,242.283,-60.621,-176.993,6.369,148.267
C01586=1223.909,242.035,-60.594,-176.995,6.367,148.267
C01587=1223.914,241.787,-60.568,-176.998,6.365,148.268
C01588=1223.918,241.538,-60.542,-177.000,6.363,148.268
C01589=1223.922,241.289,-60.517,-177.003,6.361,148.268
C01590=1223.927,241.041,-60.490,-177.005,6.359,148.268
C01591=1223.931,240.792,-60.464,-177.008,6.357,148.269
C01592=1223.936,240.544,-60.439,-177.010,6.355,148.269
C01593=1223.940,240.295,-60.413,-177.013,6.353,148.269
C01594=1223.945,240.047,-60.386,-177.015,6.351,148.269
C01595=1223.949,239.798,-60.360,-177.018,6.349,148.270
C01596=1223.953,239.549,-60.334,-177.021,6.347,148.270
C01597=1223.958,239.301,-60.309,-177.023,6.345,148.270
C01598=1223.963,239.052,-60.283,-177.025,6.343,148.270
C01599=1223.967,238.803,-60.257,-177.028,6.341,148.271
C01600=1223.971,238.554,-60.231,-177.031,6.340,148.271
C01601=1223.976,238.307,-60.205,-177.033,6.338,148.271
C01602=1223.980,238.058,-60.179,-177.036,6.336,148.272
C01603=1223.986,237.786,-60.151,-177.039,6.334,148.272
C01604=1223.991,237.514,-60.123,-177.041,6.332,148.272
C01605=1223.995,237.243,-60.094,-177.044,6.329,148.273
C01606=1224.000,236.972,-60.066,-177.047,6.327,148.273
C01607=1224.005,236.723,-60.041,-177.049,6.325,148.273
C01608=1224.009,236.474,-60.015,-177.052,6.323,148.273
C01609=1224.013,236.225,-59.989,-177.054,6.322,148.274
C01610=1224.018,235.977,-59.964,-177.057,6.320,148.274
C01611=1224.022,235.729,-59.938,-177.060,6.318,148.274
C01612=1224.026,235.480,-59.912,-177.062,6.316,148.275
C01613=1224.032,235.231,-59.886,-177.064,6.314,148.275
C01614=1224.036,234.983,-59.861,-177.067,6.312,148.275
C01615=1224.040,234.734,-59.835,-177.070,6.310,148.275
C01616=1224.045,234.485,-59.809,-177.072,6.308,148.276
C01617=1224.050,234.237,-59.784,-177.075,6.306,148.276
C01618=1224.054,233.988,-59.758,-177.077,6.304,148.276
C01619=1224.058,233.739,-59.732,-177.080,6.302,148.276
C01620=1224.063,233.491,-59.707,-177.082,6.300,148.277
C01621=1224.067,233.242,-59.681,-177.085,6.298,148.277
C01622=1224.072,232.993,-59.656,-177.087,6.297,148.277
C01623=1224.076,232.745,-59.631,-177.090,6.296,148.278
C01624=1224.081,232.496,-59.605,-177.092,6.294,148.278
C01625=1224.085,232.248,-59.579,-177.095,6.292,148.278
C01626=1224.090,231.999,-59.554,-177.097,6.290,148.279
C01627=1224.094,231.750,-59.528,-177.100,6.288,148.279
C01628=1224.099,231.502,-59.503,-177.102,6.286,148.279
C01629=1224.103,231.253,-59.478,-177.105,6.284,148.279
C01630=1224.107,231.004,-59.452,-177.107,6.282,148.280
C01631=1224.112,230.756,-59.426,-177.110,6.280,148.280
C01632=1224.117,230.507,-59.401,-177.113,6.278,148.280
C01633=1224.122,230.258,-59.376,-177.115,6.277,148.281
C01634=1224.126,230.010,-59.350,-177.118,6.275,148.281
C01635=1224.130,229.761,-59.324,-177.120,6.273,148.281
C01636=1224.135,229.513,-59.299,-177.123,6.271,148.281
C01637=1224.139,229.263,-59.274,-177.125,6.269,148.282
C01638=1224.144,229.015,-59.249,-177.128,6.267,148.282
C01639=1224.148,228.766,-59.223,-177.131,6.265,148.282
C01640=1224.153,228.517,-59.198,-177.133,6.263,148.283
C01641=1224.158,228.269,-59.173,-177.136,6.261,148.283
C01642=1224.161,228.020,-59.147,-177.138,6.259,148.283
C01643=1224.166,227.772,-59.123,-177.141,6.258,148.284
C01644=1224.171,227.523,-59.097,-177.143,6.256,148.284
C01645=1224.176,227.275,-59.072,-177.145,6.254,148.284
C01646=1224.180,227.025,-59.047,-177.148,6.253,148.285
C01647=1224.185,226.777,-59.021,-177.150,6.251,148.285
C01648=1224.189,226.528,-58.996,-177.153,6.249,148.285
C01649=1224.193,226.279,-58.971,-177.156,6.247,148.285
C01650=1224.198,226.031,-58.946,-177.158,6.245,148.286
C01651=1224.202,225.782,-58.921,-177.161,6.243,148.286
C01652=1224.207,225.534,-58.895,-177.164,6.241,148.286
C01653=1224.212,225.284,-58.870,-177.166,6.239,148.287
C01654=1224.216,225.036,-58.845,-177.169,6.238,148.287
C01655=1224.220,224.787,-58.820,-177.171,6.236,148.287
C01656=1224.225,224.539,-58.795,-177.174,6.234,148.288
C01657=1224.230,224.289,-58.770,-177.176,6.232,148.288
C01658=1224.234,224.041,-58.744,-177.179,6.230,148.288
C01659=1224.239,223.792,-58.719,-177.181,6.229,148.289
C01660=1224.243,223.544,-58.695,-177.184,6.227,148.289
C01661=1224.248,223.295,-58.670,-177.186,6.225,148.289
C01662=1224.252,223.047,-58.644,-177.189,6.223,148.290
C01663=1224.257,222.797,-58.619,-177.191,6.221,148.290
C01664=1224.261,222.549,-58.594,-177.194,6.220,148.290
C01665=1224.266,222.300,-58.569,-177.197,6.218,148.291
C01666=1224.271,222.051,-58.545,-177.199,6.216,148.291
C01667=1224.275,221.803,-58.520,-177.202,6.214,148.291
C01668=1224.279,221.554,-58.495,-177.205,6.212,148.291
C01669=1224.284,221.305,-58.470,-177.207,6.210,148.292
C01670=1224.288,221.057,-58.445,-177.210,6.208,148.292
C01671=1224.293,220.808,-58.420,-177.212,6.207,148.293
C01672=1224.297,220.559,-58.395,-177.215,6.205,148.293
C01673=1224.302,220.310,-58.370,-177.217,6.204,148.293
C01674=1224.306,220.061,-58.346,-177.220,6.202,148.293
C01675=1224.311,219.813,-58.321,-177.222,6.200,148.294
C01676=1224.315,219.565,-58.296,-177.225,6.198,148.294
C01677=1224.320,219.315,-58.271,-177.227,6.196,148.294
C01678=1224.325,219.067,-58.246,-177.230,6.194,148.295
C01679=1224.329,218.818,-58.221,-177.232,6.192,148.295
C01680=1224.334,218.569,-58.197,-177.235,6.190,148.295
C01681=1224.339,218.321,-58.172,-177.238,6.188,148.296
C01682=1224.343,218.072,-58.147,-177.240,6.187,148.296
C01683=1224.347,217.824,-58.122,-177.242,6.186,148.296
C01684=1224.351,217.574,-58.098,-177.245,6.184,148.297
C01685=1224.356,217.326,-58.073,-177.248,6.182,148.297
C01686=1224.361,217.077,-58.048,-177.250,6.180,148.297
C01687=1224.365,216.828,-58.024,-177.253,6.178,148.298
C01688=1224.370,216.579,-57.999,-177.256,6.176,148.298
C01689=1224.375,216.331,-57.974,-177.258,6.174,148.298
C01690=1224.379,216.082,-57.949,-177.261,6.172,148.299
C01691=1224.383,215.834,-57.925,-177.263,6.171,148.299
C01692=1224.388,215.584,-57.900,-177.266,6.170,148.299
C01693=1224.392,215.336,-57.876,-177.268,6.168,148.300
C01694=1224.397,215.087,-57.851,-177.271,6.166,148.300
C01695=1224.401,214.838,-57.827,-177.273,6.164,148.300
C01696=1224.406,214.589,-57.802,-177.276,6.162,148.301
C01697=1224.411,214.341,-57.778,-177.279,6.160,148.301
C01698=1224.416,214.093,-57.753,-177.281,6.158,148.301
C01699=1224.419,213.843,-57.728,-177.284,6.157,148.302
C01700=1224.425,213.595,-57.704,-177.286,6.156,148.302
C01701=1224.429,213.346,-57.680,-177.289,6.154,148.302
C01702=1224.433,213.097,-57.655,-177.291,6.152,148.303
C01703=1224.438,212.849,-57.631,-177.294,6.150,148.303
C01704=1224.443,212.600,-57.606,-177.297,6.148,148.303
C01705=1224.447,212.351,-57.581,-177.299,6.146,148.304
C01706=1224.452,212.102,-57.557,-177.302,6.144,148.304
C01707=1224.457,211.831,-57.531,-177.305,6.143,148.305
C01708=1224.462,211.561,-57.505,-177.308,6.141,148.305
C01709=1224.466,211.290,-57.478,-177.310,6.139,148.305
C01710=1224.472,211.020,-57.451,-177.313,6.137,148.306
C01711=1224.476,210.772,-57.427,-177.315,6.136,148.306
C01712=1224.481,210.523,-57.403,-177.318,6.134,148.306
C01713=1224.485,210.273,-57.378,-177.321,6.132,148.307
C01714=1224.490,210.025,-57.354,-177.323,6.130,148.307
C01715=1224.495,209.776,-57.330,-177.325,6.129,148.307
C01716=1224.499,209.528,-57.306,-177.328,6.127,148.308
C01717=1224.503,209.279,-57.282,-177.331,6.125,148.308
C01718=1224.508,209.030,-57.257,-177.334,6.124,148.308
C01719=1224.513,208.781,-57.233,-177.336,6.122,148.309
C01720=1224.517,208.533,-57.209,-177.339,6.120,148.309
C01721=1224.522,208.284,-57.184,-177.341,6.119,148.309
C01722=1224.526,208.035,-57.160,-177.344,6.117,148.310
C01723=1224.530,207.786,-57.136,-177.346,6.115,148.310
C01724=1224.536,207.537,-57.112,-177.349,6.113,148.310
C01725=1224.540,207.289,-57.088,-177.352,6.112,148.311
C01726=1224.545,207.040,-57.064,-177.354,6.110,148.311
C01727=1224.549,206.791,-57.039,-177.356,6.109,148.312
C01728=1224.554,206.542,-57.015,-177.359,6.107,148.312
C01729=1224.558,206.293,-56.991,-177.362,6.105,148.312
C01730=1224.563,206.045,-56.967,-177.364,6.103,148.313
C01731=1224.568,205.796,-56.943,-177.367,6.101,148.313
C01732=1224.572,205.547,-56.919,-177.370,6.099,148.313
C01733=1224.576,205.298,-56.895,-177.372,6.098,148.314
C01734=1224.581,205.050,-56.871,-177.374,6.097,148.314
C01735=1224.586,204.800,-56.847,-177.377,6.095,148.314
C01736=1224.590,204.552,-56.823,-177.380,6.093,148.315
C01737=1224.595,204.303,-56.799,-177.383,6.091,148.315
C01738=1224.600,204.054,-56.775,-177.385,6.089,148.316
C01739=1224.604,203.806,-56.751,-177.387,6.088,148.316
C01740=1224.609,203.556,-56.727,-177.390,6.087,148.316
C01741=1224.613,203.308,-56.703,-177.393,6.085,148.317
C01742=1224.618,203.059,-56.679,-177.395,6.083,148.317
C01743=1224.622,202.810,-56.655,-177.398,6.081,148.317
C01744=1224.627,202.562,-56.631,-177.400,6.080,148.318
C01745=1224.631,202.313,-56.608,-177.403,6.078,148.318
C01746=1224.636,202.064,-56.584,-177.405,6.076,148.318
C01747=1224.641,201.815,-56.560,-177.408,6.074,148.319
C01748=1224.645,201.566,-56.535,-177.411,6.073,148.319
C01749=1224.650,201.317,-56.512,-177.413,6.072,148.320
C01750=1224.654,201.068,-56.488,-177.416,6.070,148.320
C01751=1224.659,200.819,-56.465,-177.419,6.068,148.320
C01752=1224.663,200.571,-56.441,-177.421,6.066,148.321
C01753=1224.668,200.322,-56.417,-177.424,6.065,148.321
C01754=1224.672,200.073,-56.393,-177.426,6.064,148.321
C01755=1224.677,199.824,-56.370,-177.429,6.062,148.322
C01756=1224.682,199.576,-56.345,-177.431,6.060,148.322
C01757=1224.687,199.327,-56.322,-177.434,6.058,148.322
C01758=1224.692,199.078,-56.298,-177.436,6.057,148.323
C01759=1224.696,198.829,-56.274,-177.439,6.055,148.323
C01760=1224.701,198.580,-56.251,-177.442,6.054,148.324
C01761=1224.705,198.332,-56.227,-177.444,6.052,148.324
C01762=1224.710,198.083,-56.204,-177.447,6.050,148.324
C01763=1224.714,197.834,-56.180,-177.449,6.049,148.325
C01764=1224.718,197.585,-56.156,-177.452,6.047,148.325
C01765=1224.723,197.336,-56.132,-177.454,6.045,148.325
C01766=1224.728,197.086,-56.109,-177.457,6.043,148.326
C01767=1224.732,196.838,-56.085,-177.459,6.042,148.326
C01768=1224.737,196.589,-56.062,-177.462,6.041,148.327
C01769=1224.741,196.340,-56.038,-177.465,6.039,148.327
C01770=1224.746,196.092,-56.014,-177.467,6.037,148.327
C01771=1224.750,195.843,-55.991,-177.469,6.036,148.328
C01772=1224.755,195.594,-55.967,-177.472,6.034,148.328
C01773=1224.760,195.345,-55.944,-177.475,6.032,148.328
C01774=1224.764,195.096,-55.920,-177.477,6.031,148.329
C01775=1224.769,194.847,-55.897,-177.480,6.030,148.329
C01776=1224.774,194.599,-55.874,-177.483,6.028,148.330
C01777=1224.778,194.350,-55.851,-177.485,6.026,148.330
C01778=1224.783,194.102,-55.827,-177.488,6.024,148.330
C01779=1224.787,193.853,-55.803,-177.490,6.023,148.331
C01780=1224.792,193.604,-55.780,-177.493,6.022,148.331
C01781=1224.797,193.355,-55.757,-177.495,6.020,148.331
C01782=1224.801,193.105,-55.733,-177.498,6.018,148.332
C01783=1224.806,192.856,-55.710,-177.501,6.017,148.332
C01784=1224.811,192.608,-55.686,-177.503,6.015,148.333
C01785=1224.815,192.359,-55.663,-177.506,6.013,148.333
C01786=1224.820,192.110,-55.639,-177.508,6.012,148.333
C01787=1224.824,191.861,-55.616,-177.511,6.011,148.334
C01788=1224.829,191.612,-55.593,-177.513,6.009,148.334
C01789=1224.833,191.363,-55.570,-177.516,6.007,148.334
C01790=1224.838,191.114,-55.546,-177.519,6.005,148.335
C01791=1224.843,190.865,-55.523,-177.521,6.004,148.335
C01792=1224.848,190.617,-55.500,-177.524,6.003,148.336
C01793=1224.852,190.368,-55.477,-177.526,6.001,148.336
C01794=1224.857,190.119,-55.454,-177.528,6.000,148.337
C01795=1224.861,189.870,-55.431,-177.531,5.998,148.337
C01796=1224.866,189.621,-55.407,-177.534,5.996,148.337
C01797=1224.871,189.372,-55.384,-177.537,5.995,148.338
C01798=1224.875,189.123,-55.361,-177.539,5.994,148.338
C01799=1224.879,188.874,-55.338,-177.542,5.992,148.339
C01800=1224.884,188.625,-55.314,-177.544,5.990,148.339
C01801=1224.889,188.377,-55.291,-177.546,5.989,148.339
C01802=1224.893,188.128,-55.269,-177.549,5.987,148.340
C01803=1224.898,187.879,-55.245,-177.552,5.985,148.340
C01804=1224.903,187.630,-55.222,-177.555,5.984,148.341
C01805=1224.907,187.381,-55.199,-177.557,5.983,148.341
C01806=1224.911,187.132,-55.176,-177.559,5.981,148.341
C01807=1224.916,186.883,-55.152,-177.562,5.979,148.342
C01808=1224.921,186.635,-55.129,-177.565,5.978,148.342
C01809=1224.926,186.386,-55.106,-177.567,5.976,148.343
